REGION Network 138: CIP Line Blending Cluster 1 Request
   RUNG wire#powerrail
      Contact( "AlwaysTRUE" )
      wire#w1
      Contact( "General_Blend".Blend_Cluster1.CIP_Line1."CIP Enable" )
      Contact( "General_Blend".Blend_Cluster1.CIP_Line1."CIP Request" )
      Contact( "THE2_From_BT_To_Mixing".CIPEnable )
      wire#w2
      Coil( "Mix_to_CIP".CIP_Request."Blending Cluster 1".Blending_Cluster1_LineProduct_Request )
   END_RUNG
   RUNG wire#w1
      Contact( "General_Blend".Blend_Cluster1.CIP_Line2."CIP Enable" )
      Contact( "General_Blend".Blend_Cluster1.CIP_Line2."CIP Request" )
      Contact( "THE1_From_BT_To_Mixing".CIPEnable )
   END_RUNG wire#w2
   RUNG wire#w1
      Contact( "General_Blend".Blend_Cluster1.CIP_Line3."CIP Enable" )
      Contact( "General_Blend".Blend_Cluster1.CIP_Line3."CIP Request" )
      Contact( "General Buffer"."CIP Enable".Cluster1_Line3 )
   END_RUNG wire#w2
   // the same network as SCL:
   "Mix_to_CIP".CIP_Request."Blending Cluster 1".Blending_Cluster1_LineProduct_Request := "AlwaysTRUE" AND (("General_Blend".Blend_Cluster1.CIP_Line1."CIP Enable" AND "General_Blend".Blend_Cluster1.CIP_Line1."CIP Request" AND "THE2_From_BT_To_Mixing".CIPEnable) OR ("General_Blend".Blend_Cluster1.CIP_Line2."CIP Enable" AND "General_Blend".Blend_Cluster1.CIP_Line2."CIP Request" AND "THE1_From_BT_To_Mixing".CIPEnable) OR ("General_Blend".Blend_Cluster1.CIP_Line3."CIP Enable" AND "General_Blend".Blend_Cluster1.CIP_Line3."CIP Request" AND "General Buffer"."CIP Enable".Cluster1_Line3));
END_REGION

REGION Network 139: CIP Line Blending Cluster 1 Line OK
   RUNG wire#powerrail
      Contact( "AlwaysTRUE" )
      wire#w1
      Contact( "General_Blend".Blend_Cluster1.CIP_Line1."CIP Request" )
      Contact( "IO_Valve_Buffer_DB"."AV-22.11".FB_OPEN )
      Contact( "IO_Valve_Blend30_DB"."AV-30.12".FB_OPEN )
      wire#w2
      Contact( "IO_Valve_Blend30_DB"."AV-30.13".FB_OPEN )
      wire#w3
      Contact( "THE2_From_BT_To_Mixing".LineCIP_Open )
      wire#w4
      Coil( "Mix_to_CIP".CIP_Line_OK."Blending Cluster 1".Blending_Cluster1_LineProduct_LineOK )
   END_RUNG
   RUNG wire#w2
      Contact( "IO_Valve_Blend30_DB"."AV-30.14".FB_OPEN )
   END_RUNG wire#w3
   RUNG wire#w1
      Contact( "General_Blend".Blend_Cluster1.CIP_Line2."CIP Request" )
      Contact( "IO_Valve_Buffer_DB"."AV-22.11".FB_OPEN )
      Contact( "IO_Valve_Blend30_DB"."AV-30.15".FB_OPEN )
      wire#w5
      Contact( "IO_Valve_Blend30_DB"."AV-30.16".FB_OPEN )
      wire#w6
      Contact( "THE1_From_BT_To_Mixing".LineCIP_Open )
   END_RUNG wire#w4
   RUNG wire#w5
      Contact( "IO_Valve_Blend30_DB"."AV-30.17".FB_OPEN )
   END_RUNG wire#w6
   RUNG wire#w1
      Contact( "General_Blend".Blend_Cluster1.CIP_Line3."CIP Request" )
      Contact( "IO_Valve_Buffer_DB"."AV-22.11".FB_OPEN )
      Contact( "IO_Valve_Blend30_DB"."AV-30.18".FB_OPEN )
      wire#w7
      Contact( "IO_Valve_Blend30_DB"."AV-30.19".FB_OPEN )
      wire#w8
      Contact( "General Buffer"."CIP Line Open".Cluster1_Line3 )
   END_RUNG wire#w4
   RUNG wire#w7
      Contact( "IO_Valve_Blend30_DB"."AV-30.20".FB_OPEN )
   END_RUNG wire#w8
   // the same network as SCL:
   "Mix_to_CIP".CIP_Line_OK."Blending Cluster 1".Blending_Cluster1_LineProduct_LineOK := "AlwaysTRUE" AND (("General_Blend".Blend_Cluster1.CIP_Line1."CIP Request" AND "IO_Valve_Buffer_DB"."AV-22.11".FB_OPEN AND "IO_Valve_Blend30_DB"."AV-30.12".FB_OPEN AND ("IO_Valve_Blend30_DB"."AV-30.13".FB_OPEN OR "IO_Valve_Blend30_DB"."AV-30.14".FB_OPEN) AND "THE2_From_BT_To_Mixing".LineCIP_Open) OR ("General_Blend".Blend_Cluster1.CIP_Line2."CIP Request" AND "IO_Valve_Buffer_DB"."AV-22.11".FB_OPEN AND "IO_Valve_Blend30_DB"."AV-30.15".FB_OPEN AND ("IO_Valve_Blend30_DB"."AV-30.16".FB_OPEN OR "IO_Valve_Blend30_DB"."AV-30.17".FB_OPEN) AND "THE1_From_BT_To_Mixing".LineCIP_Open) OR ("General_Blend".Blend_Cluster1.CIP_Line3."CIP Request" AND "IO_Valve_Buffer_DB"."AV-22.11".FB_OPEN AND "IO_Valve_Blend30_DB"."AV-30.18".FB_OPEN AND ("IO_Valve_Blend30_DB"."AV-30.19".FB_OPEN OR "IO_Valve_Blend30_DB"."AV-30.20".FB_OPEN) AND "General Buffer"."CIP Line Open".Cluster1_Line3));
END_REGION

REGION Network 140: CIP Line Blending Cluster 1 Valve Cmd
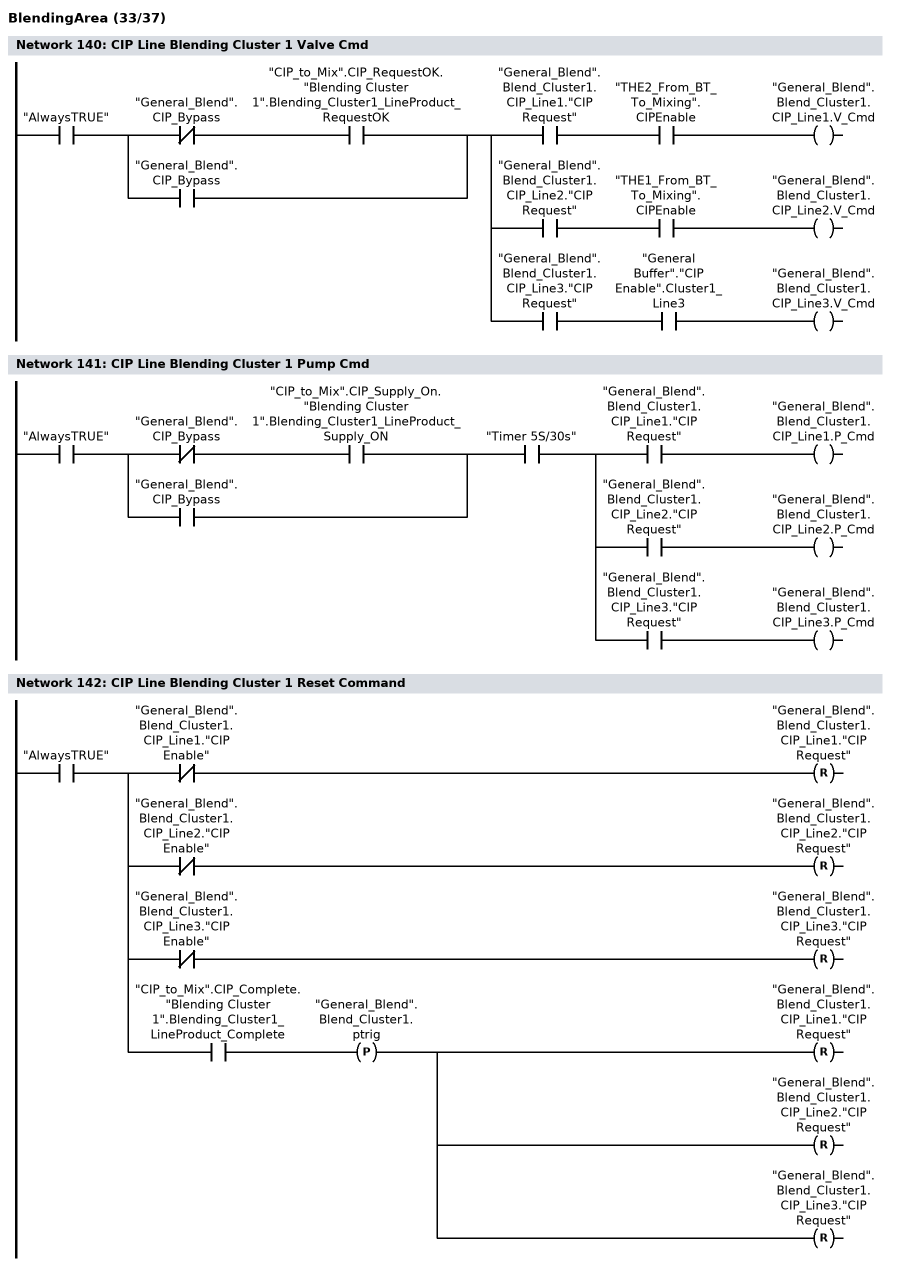
   RUNG wire#powerrail
      Contact( "AlwaysTRUE" )
      wire#w1
      I_Contact( "General_Blend".CIP_Bypass )
      Contact( "CIP_to_Mix".CIP_RequestOK."Blending Cluster 1".Blending_Cluster1_LineProduct_RequestOK )
      wire#w2
      Contact( "General_Blend".Blend_Cluster1.CIP_Line1."CIP Request" )
      Contact( "THE2_From_BT_To_Mixing".CIPEnable )
      Coil( "General_Blend".Blend_Cluster1.CIP_Line1.V_Cmd )
   END_RUNG
   RUNG wire#w1
      Contact( "General_Blend".CIP_Bypass )
   END_RUNG wire#w2
   RUNG wire#w2
      Contact( "General_Blend".Blend_Cluster1.CIP_Line2."CIP Request" )
      Contact( "THE1_From_BT_To_Mixing".CIPEnable )
      Coil( "General_Blend".Blend_Cluster1.CIP_Line2.V_Cmd )
   END_RUNG
   RUNG wire#w2
      Contact( "General_Blend".Blend_Cluster1.CIP_Line3."CIP Request" )
      Contact( "General Buffer"."CIP Enable".Cluster1_Line3 )
      Coil( "General_Blend".Blend_Cluster1.CIP_Line3.V_Cmd )
   END_RUNG
   // the same network as SCL:
   #_w1 := "AlwaysTRUE" AND ((NOT "General_Blend".CIP_Bypass AND "CIP_to_Mix".CIP_RequestOK."Blending Cluster 1".Blending_Cluster1_LineProduct_RequestOK) OR "General_Blend".CIP_Bypass);
   "General_Blend".Blend_Cluster1.CIP_Line1.V_Cmd := #_w1 AND "General_Blend".Blend_Cluster1.CIP_Line1."CIP Request" AND "THE2_From_BT_To_Mixing".CIPEnable;
   "General_Blend".Blend_Cluster1.CIP_Line2.V_Cmd := #_w1 AND "General_Blend".Blend_Cluster1.CIP_Line2."CIP Request" AND "THE1_From_BT_To_Mixing".CIPEnable;
   "General_Blend".Blend_Cluster1.CIP_Line3.V_Cmd := #_w1 AND "General_Blend".Blend_Cluster1.CIP_Line3."CIP Request" AND "General Buffer"."CIP Enable".Cluster1_Line3;
END_REGION

REGION Network 141: CIP Line Blending Cluster 1 Pump Cmd
   RUNG wire#powerrail
      Contact( "AlwaysTRUE" )
      wire#w1
      I_Contact( "General_Blend".CIP_Bypass )
      Contact( "CIP_to_Mix".CIP_Supply_On."Blending Cluster 1".Blending_Cluster1_LineProduct_Supply_ON )
      wire#w2
      Contact( "Timer 5S/30s" )
      wire#w3
      Contact( "General_Blend".Blend_Cluster1.CIP_Line1."CIP Request" )
      Coil( "General_Blend".Blend_Cluster1.CIP_Line1.P_Cmd )
   END_RUNG
   RUNG wire#w1
      Contact( "General_Blend".CIP_Bypass )
   END_RUNG wire#w2
   RUNG wire#w3
      Contact( "General_Blend".Blend_Cluster1.CIP_Line2."CIP Request" )
      Coil( "General_Blend".Blend_Cluster1.CIP_Line2.P_Cmd )
   END_RUNG
   RUNG wire#w3
      Contact( "General_Blend".Blend_Cluster1.CIP_Line3."CIP Request" )
      Coil( "General_Blend".Blend_Cluster1.CIP_Line3.P_Cmd )
   END_RUNG
   // the same network as SCL:
   #_w1 := "AlwaysTRUE" AND ((NOT "General_Blend".CIP_Bypass AND "CIP_to_Mix".CIP_Supply_On."Blending Cluster 1".Blending_Cluster1_LineProduct_Supply_ON) OR "General_Blend".CIP_Bypass) AND "Timer 5S/30s";
   "General_Blend".Blend_Cluster1.CIP_Line1.P_Cmd := #_w1 AND "General_Blend".Blend_Cluster1.CIP_Line1."CIP Request";
   "General_Blend".Blend_Cluster1.CIP_Line2.P_Cmd := #_w1 AND "General_Blend".Blend_Cluster1.CIP_Line2."CIP Request";
   "General_Blend".Blend_Cluster1.CIP_Line3.P_Cmd := #_w1 AND "General_Blend".Blend_Cluster1.CIP_Line3."CIP Request";
END_REGION

REGION Network 142: CIP Line Blending Cluster 1 Reset Command
   RUNG wire#powerrail
      Contact( "AlwaysTRUE" )
      wire#w1
      I_Contact( "General_Blend".Blend_Cluster1.CIP_Line1."CIP Enable" )
      R_Coil( "General_Blend".Blend_Cluster1.CIP_Line1."CIP Request" )
   END_RUNG
   RUNG wire#w1
      I_Contact( "General_Blend".Blend_Cluster1.CIP_Line2."CIP Enable" )
      R_Coil( "General_Blend".Blend_Cluster1.CIP_Line2."CIP Request" )
   END_RUNG
   RUNG wire#w1
      I_Contact( "General_Blend".Blend_Cluster1.CIP_Line3."CIP Enable" )
      R_Coil( "General_Blend".Blend_Cluster1.CIP_Line3."CIP Request" )
   END_RUNG
   RUNG wire#w1
      Contact( "CIP_to_Mix".CIP_Complete."Blending Cluster 1".Blending_Cluster1_LineProduct_Complete )
      P_Trig( "General_Blend".Blend_Cluster1.ptrig )
      wire#w2
      R_Coil( "General_Blend".Blend_Cluster1.CIP_Line1."CIP Request" )
   END_RUNG
   RUNG wire#w2
      R_Coil( "General_Blend".Blend_Cluster1.CIP_Line2."CIP Request" )
   END_RUNG
   RUNG wire#w2
      R_Coil( "General_Blend".Blend_Cluster1.CIP_Line3."CIP Request" )
   END_RUNG
   // the same network as SCL:
   IF "AlwaysTRUE" AND NOT "General_Blend".Blend_Cluster1.CIP_Line1."CIP Enable" THEN
       "General_Blend".Blend_Cluster1.CIP_Line1."CIP Request" := FALSE;
   END_IF;
   IF "AlwaysTRUE" AND NOT "General_Blend".Blend_Cluster1.CIP_Line2."CIP Enable" THEN
       "General_Blend".Blend_Cluster1.CIP_Line2."CIP Request" := FALSE;
   END_IF;
   IF "AlwaysTRUE" AND NOT "General_Blend".Blend_Cluster1.CIP_Line3."CIP Enable" THEN
       "General_Blend".Blend_Cluster1.CIP_Line3."CIP Request" := FALSE;
   END_IF;
   #_w1 := "AlwaysTRUE" AND "CIP_to_Mix".CIP_Complete."Blending Cluster 1".Blending_Cluster1_LineProduct_Complete;
   #_w2 := #_w1 AND NOT "General_Blend".Blend_Cluster1.ptrig;   // rising edge
   "General_Blend".Blend_Cluster1.ptrig := #_w1;
   IF #_w2 THEN
       "General_Blend".Blend_Cluster1.CIP_Line1."CIP Request" := FALSE;
       "General_Blend".Blend_Cluster1.CIP_Line2."CIP Request" := FALSE;
       "General_Blend".Blend_Cluster1.CIP_Line3."CIP Request" := FALSE;
   END_IF;
END_REGION

REGION Network 144: CIP Line Blending Cluster 2 Enable
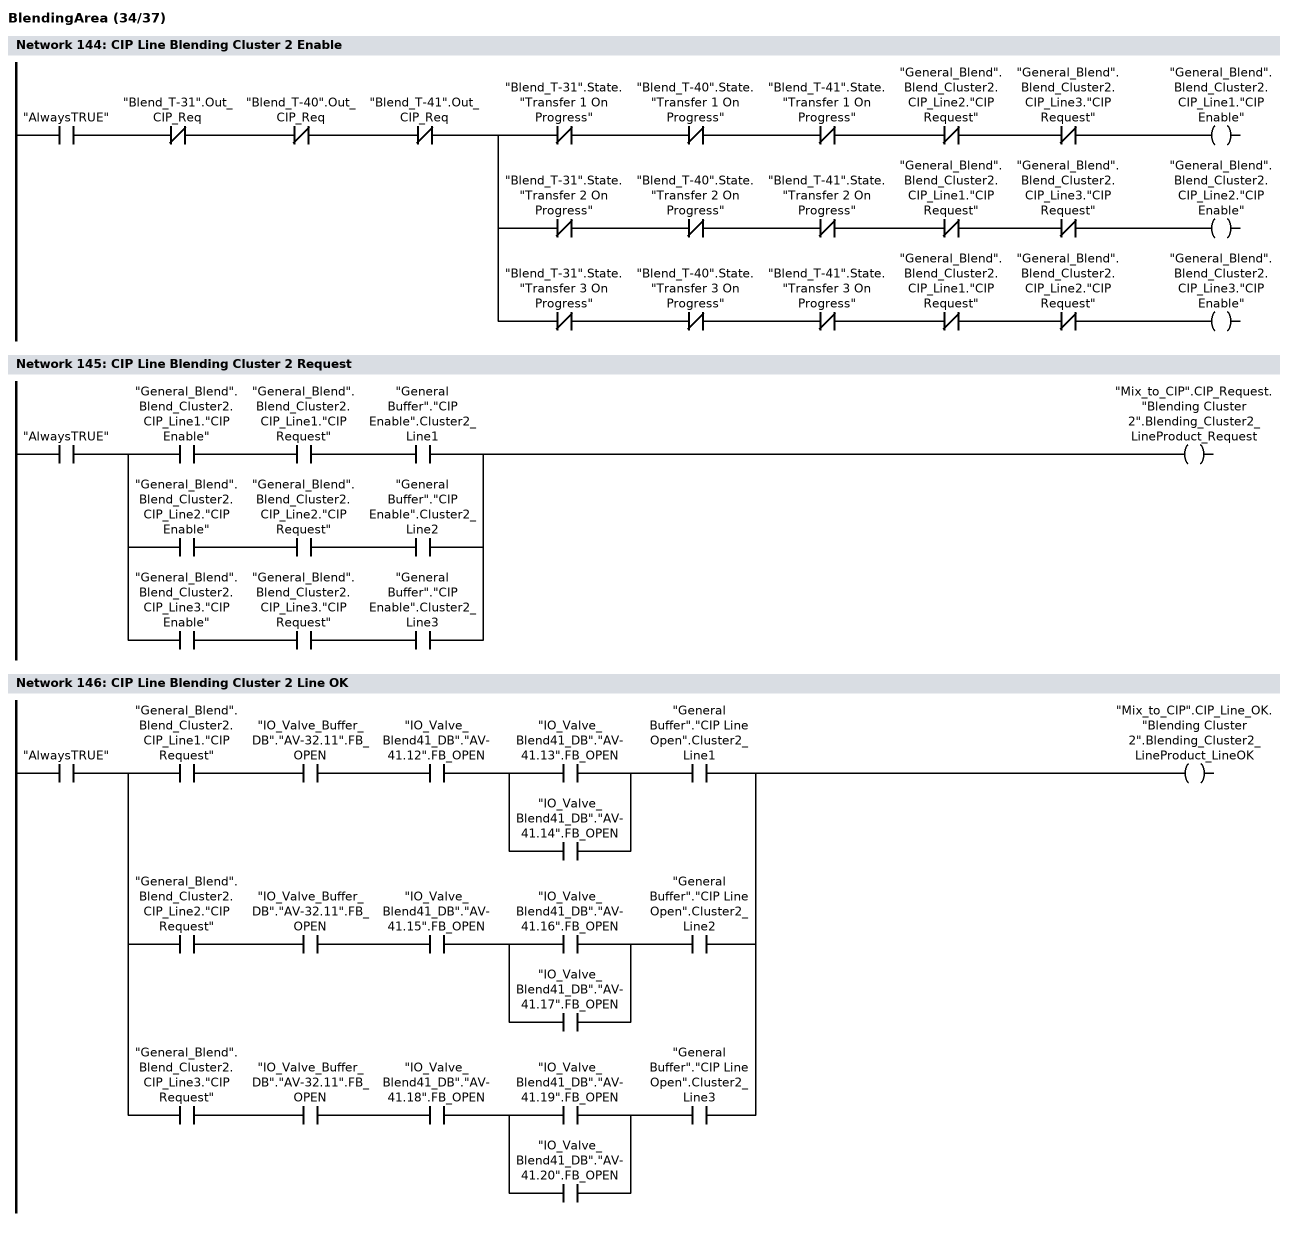
   RUNG wire#powerrail
      Contact( "AlwaysTRUE" )
      I_Contact( "Blend_T-31".Out_CIP_Req )
      I_Contact( "Blend_T-40".Out_CIP_Req )
      I_Contact( "Blend_T-41".Out_CIP_Req )
      wire#w1
      I_Contact( "Blend_T-31".State."Transfer 1 On Progress" )
      I_Contact( "Blend_T-40".State."Transfer 1 On Progress" )
      I_Contact( "Blend_T-41".State."Transfer 1 On Progress" )
      I_Contact( "General_Blend".Blend_Cluster2.CIP_Line2."CIP Request" )
      I_Contact( "General_Blend".Blend_Cluster2.CIP_Line3."CIP Request" )
      Coil( "General_Blend".Blend_Cluster2.CIP_Line1."CIP Enable" )
   END_RUNG
   RUNG wire#w1
      I_Contact( "Blend_T-31".State."Transfer 2 On Progress" )
      I_Contact( "Blend_T-40".State."Transfer 2 On Progress" )
      I_Contact( "Blend_T-41".State."Transfer 2 On Progress" )
      I_Contact( "General_Blend".Blend_Cluster2.CIP_Line1."CIP Request" )
      I_Contact( "General_Blend".Blend_Cluster2.CIP_Line3."CIP Request" )
      Coil( "General_Blend".Blend_Cluster2.CIP_Line2."CIP Enable" )
   END_RUNG
   RUNG wire#w1
      I_Contact( "Blend_T-31".State."Transfer 3 On Progress" )
      I_Contact( "Blend_T-40".State."Transfer 3 On Progress" )
      I_Contact( "Blend_T-41".State."Transfer 3 On Progress" )
      I_Contact( "General_Blend".Blend_Cluster2.CIP_Line1."CIP Request" )
      I_Contact( "General_Blend".Blend_Cluster2.CIP_Line2."CIP Request" )
      Coil( "General_Blend".Blend_Cluster2.CIP_Line3."CIP Enable" )
   END_RUNG
   // the same network as SCL:
   #_w1 := "AlwaysTRUE" AND NOT "Blend_T-31".Out_CIP_Req AND NOT "Blend_T-40".Out_CIP_Req AND NOT "Blend_T-41".Out_CIP_Req;
   "General_Blend".Blend_Cluster2.CIP_Line1."CIP Enable" := #_w1 AND NOT "Blend_T-31".State."Transfer 1 On Progress" AND NOT "Blend_T-40".State."Transfer 1 On Progress" AND NOT "Blend_T-41".State."Transfer 1 On Progress" AND NOT "General_Blend".Blend_Cluster2.CIP_Line2."CIP Request" AND NOT "General_Blend".Blend_Cluster2.CIP_Line3."CIP Request";
   "General_Blend".Blend_Cluster2.CIP_Line2."CIP Enable" := #_w1 AND NOT "Blend_T-31".State."Transfer 2 On Progress" AND NOT "Blend_T-40".State."Transfer 2 On Progress" AND NOT "Blend_T-41".State."Transfer 2 On Progress" AND NOT "General_Blend".Blend_Cluster2.CIP_Line1."CIP Request" AND NOT "General_Blend".Blend_Cluster2.CIP_Line3."CIP Request";
   "General_Blend".Blend_Cluster2.CIP_Line3."CIP Enable" := #_w1 AND NOT "Blend_T-31".State."Transfer 3 On Progress" AND NOT "Blend_T-40".State."Transfer 3 On Progress" AND NOT "Blend_T-41".State."Transfer 3 On Progress" AND NOT "General_Blend".Blend_Cluster2.CIP_Line1."CIP Request" AND NOT "General_Blend".Blend_Cluster2.CIP_Line2."CIP Request";
END_REGION

REGION Network 145: CIP Line Blending Cluster 2 Request
   RUNG wire#powerrail
      Contact( "AlwaysTRUE" )
      wire#w1
      Contact( "General_Blend".Blend_Cluster2.CIP_Line1."CIP Enable" )
      Contact( "General_Blend".Blend_Cluster2.CIP_Line1."CIP Request" )
      Contact( "General Buffer"."CIP Enable".Cluster2_Line1 )
      wire#w2
      Coil( "Mix_to_CIP".CIP_Request."Blending Cluster 2".Blending_Cluster2_LineProduct_Request )
   END_RUNG
   RUNG wire#w1
      Contact( "General_Blend".Blend_Cluster2.CIP_Line2."CIP Enable" )
      Contact( "General_Blend".Blend_Cluster2.CIP_Line2."CIP Request" )
      Contact( "General Buffer"."CIP Enable".Cluster2_Line2 )
   END_RUNG wire#w2
   RUNG wire#w1
      Contact( "General_Blend".Blend_Cluster2.CIP_Line3."CIP Enable" )
      Contact( "General_Blend".Blend_Cluster2.CIP_Line3."CIP Request" )
      Contact( "General Buffer"."CIP Enable".Cluster2_Line3 )
   END_RUNG wire#w2
   // the same network as SCL:
   "Mix_to_CIP".CIP_Request."Blending Cluster 2".Blending_Cluster2_LineProduct_Request := "AlwaysTRUE" AND (("General_Blend".Blend_Cluster2.CIP_Line1."CIP Enable" AND "General_Blend".Blend_Cluster2.CIP_Line1."CIP Request" AND "General Buffer"."CIP Enable".Cluster2_Line1) OR ("General_Blend".Blend_Cluster2.CIP_Line2."CIP Enable" AND "General_Blend".Blend_Cluster2.CIP_Line2."CIP Request" AND "General Buffer"."CIP Enable".Cluster2_Line2) OR ("General_Blend".Blend_Cluster2.CIP_Line3."CIP Enable" AND "General_Blend".Blend_Cluster2.CIP_Line3."CIP Request" AND "General Buffer"."CIP Enable".Cluster2_Line3));
END_REGION

REGION Network 146: CIP Line Blending Cluster 2 Line OK
   RUNG wire#powerrail
      Contact( "AlwaysTRUE" )
      wire#w1
      Contact( "General_Blend".Blend_Cluster2.CIP_Line1."CIP Request" )
      Contact( "IO_Valve_Buffer_DB"."AV-32.11".FB_OPEN )
      Contact( "IO_Valve_Blend41_DB"."AV-41.12".FB_OPEN )
      wire#w2
      Contact( "IO_Valve_Blend41_DB"."AV-41.13".FB_OPEN )
      wire#w3
      Contact( "General Buffer"."CIP Line Open".Cluster2_Line1 )
      wire#w4
      Coil( "Mix_to_CIP".CIP_Line_OK."Blending Cluster 2".Blending_Cluster2_LineProduct_LineOK )
   END_RUNG
   RUNG wire#w2
      Contact( "IO_Valve_Blend41_DB"."AV-41.14".FB_OPEN )
   END_RUNG wire#w3
   RUNG wire#w1
      Contact( "General_Blend".Blend_Cluster2.CIP_Line2."CIP Request" )
      Contact( "IO_Valve_Buffer_DB"."AV-32.11".FB_OPEN )
      Contact( "IO_Valve_Blend41_DB"."AV-41.15".FB_OPEN )
      wire#w5
      Contact( "IO_Valve_Blend41_DB"."AV-41.16".FB_OPEN )
      wire#w6
      Contact( "General Buffer"."CIP Line Open".Cluster2_Line2 )
   END_RUNG wire#w4
   RUNG wire#w5
      Contact( "IO_Valve_Blend41_DB"."AV-41.17".FB_OPEN )
   END_RUNG wire#w6
   RUNG wire#w1
      Contact( "General_Blend".Blend_Cluster2.CIP_Line3."CIP Request" )
      Contact( "IO_Valve_Buffer_DB"."AV-32.11".FB_OPEN )
      Contact( "IO_Valve_Blend41_DB"."AV-41.18".FB_OPEN )
      wire#w7
      Contact( "IO_Valve_Blend41_DB"."AV-41.19".FB_OPEN )
      wire#w8
      Contact( "General Buffer"."CIP Line Open".Cluster2_Line3 )
   END_RUNG wire#w4
   RUNG wire#w7
      Contact( "IO_Valve_Blend41_DB"."AV-41.20".FB_OPEN )
   END_RUNG wire#w8
   // the same network as SCL:
   "Mix_to_CIP".CIP_Line_OK."Blending Cluster 2".Blending_Cluster2_LineProduct_LineOK := "AlwaysTRUE" AND (("General_Blend".Blend_Cluster2.CIP_Line1."CIP Request" AND "IO_Valve_Buffer_DB"."AV-32.11".FB_OPEN AND "IO_Valve_Blend41_DB"."AV-41.12".FB_OPEN AND ("IO_Valve_Blend41_DB"."AV-41.13".FB_OPEN OR "IO_Valve_Blend41_DB"."AV-41.14".FB_OPEN) AND "General Buffer"."CIP Line Open".Cluster2_Line1) OR ("General_Blend".Blend_Cluster2.CIP_Line2."CIP Request" AND "IO_Valve_Buffer_DB"."AV-32.11".FB_OPEN AND "IO_Valve_Blend41_DB"."AV-41.15".FB_OPEN AND ("IO_Valve_Blend41_DB"."AV-41.16".FB_OPEN OR "IO_Valve_Blend41_DB"."AV-41.17".FB_OPEN) AND "General Buffer"."CIP Line Open".Cluster2_Line2) OR ("General_Blend".Blend_Cluster2.CIP_Line3."CIP Request" AND "IO_Valve_Buffer_DB"."AV-32.11".FB_OPEN AND "IO_Valve_Blend41_DB"."AV-41.18".FB_OPEN AND ("IO_Valve_Blend41_DB"."AV-41.19".FB_OPEN OR "IO_Valve_Blend41_DB"."AV-41.20".FB_OPEN) AND "General Buffer"."CIP Line Open".Cluster2_Line3));
END_REGION

REGION Network 147: CIP Line Blending Cluster 2 Valve Cmd
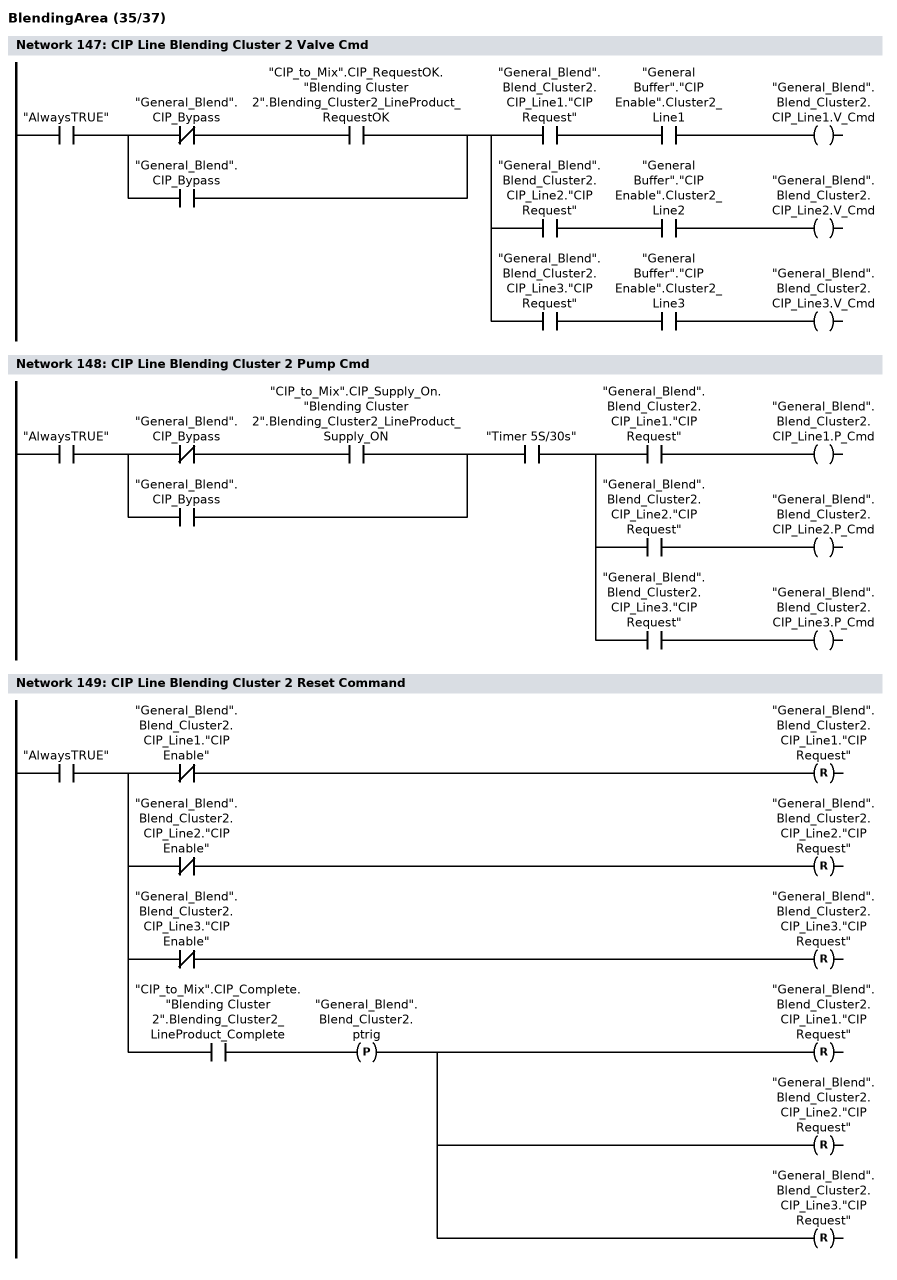
   RUNG wire#powerrail
      Contact( "AlwaysTRUE" )
      wire#w1
      I_Contact( "General_Blend".CIP_Bypass )
      Contact( "CIP_to_Mix".CIP_RequestOK."Blending Cluster 2".Blending_Cluster2_LineProduct_RequestOK )
      wire#w2
      Contact( "General_Blend".Blend_Cluster2.CIP_Line1."CIP Request" )
      Contact( "General Buffer"."CIP Enable".Cluster2_Line1 )
      Coil( "General_Blend".Blend_Cluster2.CIP_Line1.V_Cmd )
   END_RUNG
   RUNG wire#w1
      Contact( "General_Blend".CIP_Bypass )
   END_RUNG wire#w2
   RUNG wire#w2
      Contact( "General_Blend".Blend_Cluster2.CIP_Line2."CIP Request" )
      Contact( "General Buffer"."CIP Enable".Cluster2_Line2 )
      Coil( "General_Blend".Blend_Cluster2.CIP_Line2.V_Cmd )
   END_RUNG
   RUNG wire#w2
      Contact( "General_Blend".Blend_Cluster2.CIP_Line3."CIP Request" )
      Contact( "General Buffer"."CIP Enable".Cluster2_Line3 )
      Coil( "General_Blend".Blend_Cluster2.CIP_Line3.V_Cmd )
   END_RUNG
   // the same network as SCL:
   #_w1 := "AlwaysTRUE" AND ((NOT "General_Blend".CIP_Bypass AND "CIP_to_Mix".CIP_RequestOK."Blending Cluster 2".Blending_Cluster2_LineProduct_RequestOK) OR "General_Blend".CIP_Bypass);
   "General_Blend".Blend_Cluster2.CIP_Line1.V_Cmd := #_w1 AND "General_Blend".Blend_Cluster2.CIP_Line1."CIP Request" AND "General Buffer"."CIP Enable".Cluster2_Line1;
   "General_Blend".Blend_Cluster2.CIP_Line2.V_Cmd := #_w1 AND "General_Blend".Blend_Cluster2.CIP_Line2."CIP Request" AND "General Buffer"."CIP Enable".Cluster2_Line2;
   "General_Blend".Blend_Cluster2.CIP_Line3.V_Cmd := #_w1 AND "General_Blend".Blend_Cluster2.CIP_Line3."CIP Request" AND "General Buffer"."CIP Enable".Cluster2_Line3;
END_REGION

REGION Network 148: CIP Line Blending Cluster 2 Pump Cmd
   RUNG wire#powerrail
      Contact( "AlwaysTRUE" )
      wire#w1
      I_Contact( "General_Blend".CIP_Bypass )
      Contact( "CIP_to_Mix".CIP_Supply_On."Blending Cluster 2".Blending_Cluster2_LineProduct_Supply_ON )
      wire#w2
      Contact( "Timer 5S/30s" )
      wire#w3
      Contact( "General_Blend".Blend_Cluster2.CIP_Line1."CIP Request" )
      Coil( "General_Blend".Blend_Cluster2.CIP_Line1.P_Cmd )
   END_RUNG
   RUNG wire#w1
      Contact( "General_Blend".CIP_Bypass )
   END_RUNG wire#w2
   RUNG wire#w3
      Contact( "General_Blend".Blend_Cluster2.CIP_Line2."CIP Request" )
      Coil( "General_Blend".Blend_Cluster2.CIP_Line2.P_Cmd )
   END_RUNG
   RUNG wire#w3
      Contact( "General_Blend".Blend_Cluster2.CIP_Line3."CIP Request" )
      Coil( "General_Blend".Blend_Cluster2.CIP_Line3.P_Cmd )
   END_RUNG
   // the same network as SCL:
   #_w1 := "AlwaysTRUE" AND ((NOT "General_Blend".CIP_Bypass AND "CIP_to_Mix".CIP_Supply_On."Blending Cluster 2".Blending_Cluster2_LineProduct_Supply_ON) OR "General_Blend".CIP_Bypass) AND "Timer 5S/30s";
   "General_Blend".Blend_Cluster2.CIP_Line1.P_Cmd := #_w1 AND "General_Blend".Blend_Cluster2.CIP_Line1."CIP Request";
   "General_Blend".Blend_Cluster2.CIP_Line2.P_Cmd := #_w1 AND "General_Blend".Blend_Cluster2.CIP_Line2."CIP Request";
   "General_Blend".Blend_Cluster2.CIP_Line3.P_Cmd := #_w1 AND "General_Blend".Blend_Cluster2.CIP_Line3."CIP Request";
END_REGION

REGION Network 149: CIP Line Blending Cluster 2 Reset Command
   RUNG wire#powerrail
      Contact( "AlwaysTRUE" )
      wire#w1
      I_Contact( "General_Blend".Blend_Cluster2.CIP_Line1."CIP Enable" )
      R_Coil( "General_Blend".Blend_Cluster2.CIP_Line1."CIP Request" )
   END_RUNG
   RUNG wire#w1
      I_Contact( "General_Blend".Blend_Cluster2.CIP_Line2."CIP Enable" )
      R_Coil( "General_Blend".Blend_Cluster2.CIP_Line2."CIP Request" )
   END_RUNG
   RUNG wire#w1
      I_Contact( "General_Blend".Blend_Cluster2.CIP_Line3."CIP Enable" )
      R_Coil( "General_Blend".Blend_Cluster2.CIP_Line3."CIP Request" )
   END_RUNG
   RUNG wire#w1
      Contact( "CIP_to_Mix".CIP_Complete."Blending Cluster 2".Blending_Cluster2_LineProduct_Complete )
      P_Trig( "General_Blend".Blend_Cluster2.ptrig )
      wire#w2
      R_Coil( "General_Blend".Blend_Cluster2.CIP_Line1."CIP Request" )
   END_RUNG
   RUNG wire#w2
      R_Coil( "General_Blend".Blend_Cluster2.CIP_Line2."CIP Request" )
   END_RUNG
   RUNG wire#w2
      R_Coil( "General_Blend".Blend_Cluster2.CIP_Line3."CIP Request" )
   END_RUNG
   // the same network as SCL:
   IF "AlwaysTRUE" AND NOT "General_Blend".Blend_Cluster2.CIP_Line1."CIP Enable" THEN
       "General_Blend".Blend_Cluster2.CIP_Line1."CIP Request" := FALSE;
   END_IF;
   IF "AlwaysTRUE" AND NOT "General_Blend".Blend_Cluster2.CIP_Line2."CIP Enable" THEN
       "General_Blend".Blend_Cluster2.CIP_Line2."CIP Request" := FALSE;
   END_IF;
   IF "AlwaysTRUE" AND NOT "General_Blend".Blend_Cluster2.CIP_Line3."CIP Enable" THEN
       "General_Blend".Blend_Cluster2.CIP_Line3."CIP Request" := FALSE;
   END_IF;
   #_w1 := "AlwaysTRUE" AND "CIP_to_Mix".CIP_Complete."Blending Cluster 2".Blending_Cluster2_LineProduct_Complete;
   #_w2 := #_w1 AND NOT "General_Blend".Blend_Cluster2.ptrig;   // rising edge
   "General_Blend".Blend_Cluster2.ptrig := #_w1;
   IF #_w2 THEN
       "General_Blend".Blend_Cluster2.CIP_Line1."CIP Request" := FALSE;
       "General_Blend".Blend_Cluster2.CIP_Line2."CIP Request" := FALSE;
       "General_Blend".Blend_Cluster2.CIP_Line3."CIP Request" := FALSE;
   END_IF;
END_REGION

REGION Network 151: CIP to Return Line 1
   // Only for Blend Tank, Because CIP Supply from line 2 while Blend Tank can choose to return through line 1 or 2
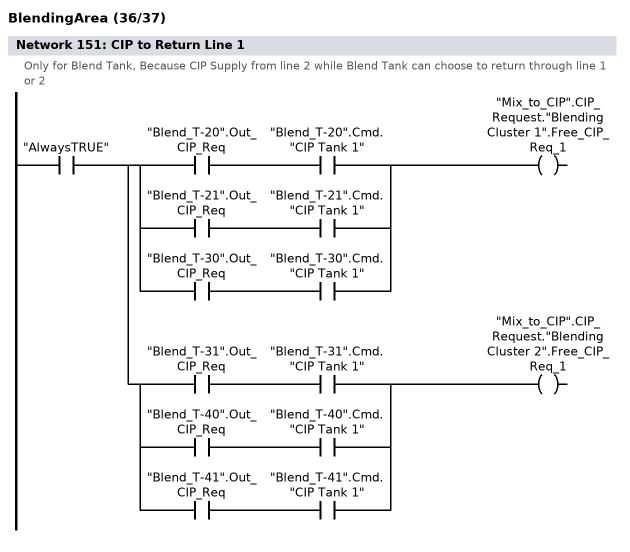
   RUNG wire#powerrail
      Contact( "AlwaysTRUE" )
      wire#w1
      Contact( "Blend_T-20".Out_CIP_Req )
      Contact( "Blend_T-20".Cmd."CIP Tank 1" )
      wire#w2
      Coil( "Mix_to_CIP".CIP_Request."Blending Cluster 1".Free_CIP_Req_1 )
   END_RUNG
   RUNG wire#w1
      Contact( "Blend_T-21".Out_CIP_Req )
      Contact( "Blend_T-21".Cmd."CIP Tank 1" )
   END_RUNG wire#w2
   RUNG wire#w1
      Contact( "Blend_T-30".Out_CIP_Req )
      Contact( "Blend_T-30".Cmd."CIP Tank 1" )
   END_RUNG wire#w2
   RUNG wire#w1
      Contact( "Blend_T-31".Out_CIP_Req )
      Contact( "Blend_T-31".Cmd."CIP Tank 1" )
      wire#w3
      Coil( "Mix_to_CIP".CIP_Request."Blending Cluster 2".Free_CIP_Req_1 )
   END_RUNG
   RUNG wire#w1
      Contact( "Blend_T-40".Out_CIP_Req )
      Contact( "Blend_T-40".Cmd."CIP Tank 1" )
   END_RUNG wire#w3
   RUNG wire#w1
      Contact( "Blend_T-41".Out_CIP_Req )
      Contact( "Blend_T-41".Cmd."CIP Tank 1" )
   END_RUNG wire#w3
   // the same network as SCL:
   "Mix_to_CIP".CIP_Request."Blending Cluster 1".Free_CIP_Req_1 := "AlwaysTRUE" AND (("Blend_T-20".Out_CIP_Req AND "Blend_T-20".Cmd."CIP Tank 1") OR ("Blend_T-21".Out_CIP_Req AND "Blend_T-21".Cmd."CIP Tank 1") OR ("Blend_T-30".Out_CIP_Req AND "Blend_T-30".Cmd."CIP Tank 1"));
   "Mix_to_CIP".CIP_Request."Blending Cluster 2".Free_CIP_Req_1 := "AlwaysTRUE" AND (("Blend_T-31".Out_CIP_Req AND "Blend_T-31".Cmd."CIP Tank 1") OR ("Blend_T-40".Out_CIP_Req AND "Blend_T-40".Cmd."CIP Tank 1") OR ("Blend_T-41".Out_CIP_Req AND "Blend_T-41".Cmd."CIP Tank 1"));
END_REGION

REGION Network 153: Valve
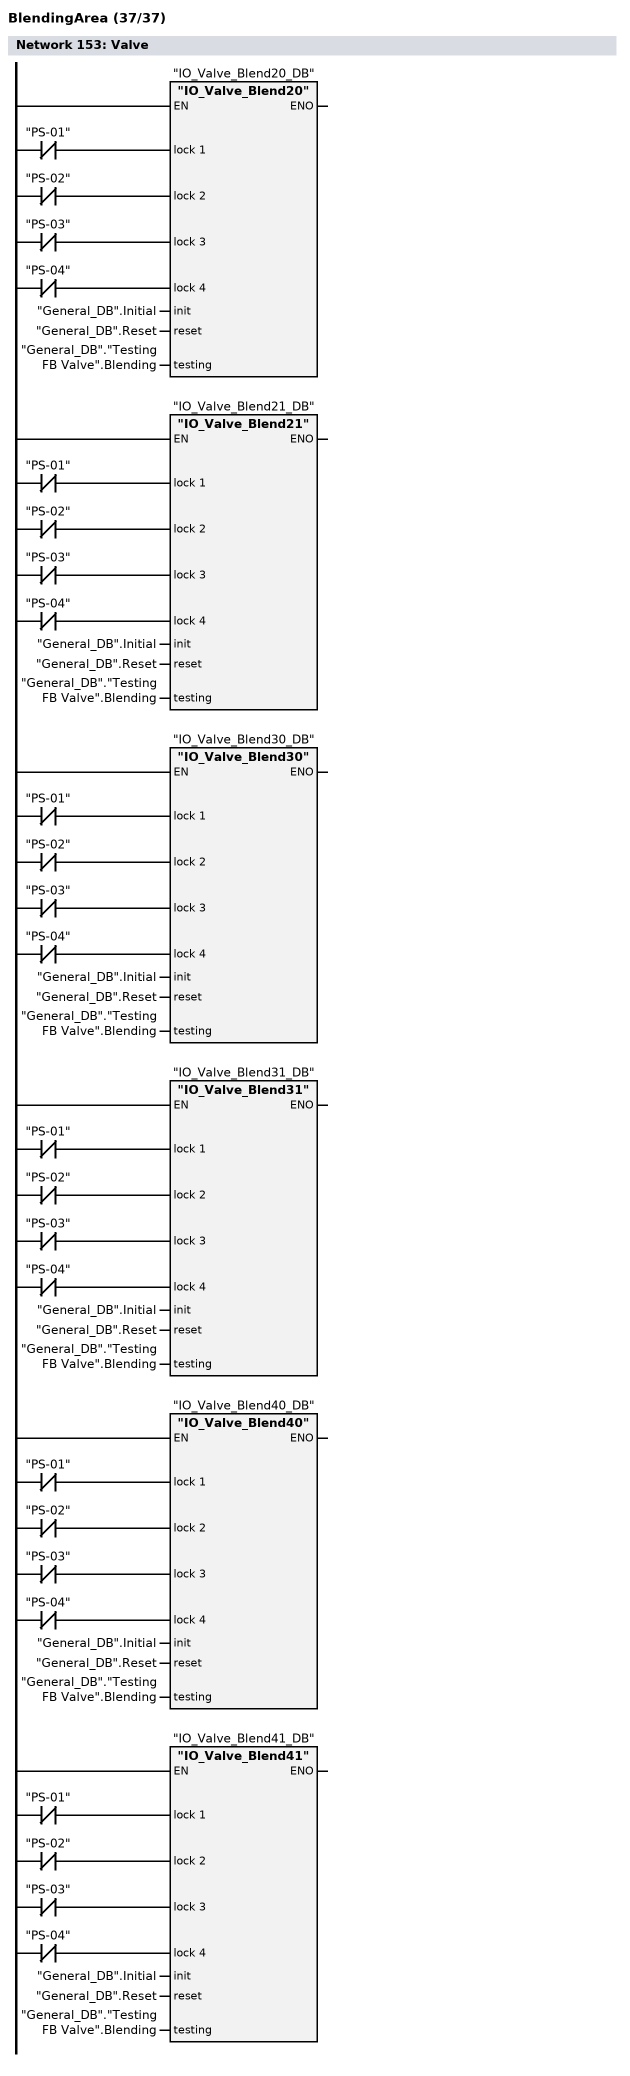
   RUNG wire#powerrail
      "IO_Valve_Blend20_DB"("lock 1" := wire#w1, "lock 2" := wire#w2, "lock 3" := wire#w3, "lock 4" := wire#w4, init := "General_DB".Initial, reset := "General_DB".Reset, testing := "General_DB"."Testing FB Valve".Blending)
   END_RUNG
   RUNG wire#powerrail
      I_Contact( "PS-01" )
   END_RUNG wire#w1
   RUNG wire#powerrail
      I_Contact( "PS-02" )
   END_RUNG wire#w2
   RUNG wire#powerrail
      I_Contact( "PS-03" )
   END_RUNG wire#w3
   RUNG wire#powerrail
      I_Contact( "PS-04" )
   END_RUNG wire#w4
   RUNG wire#powerrail
      "IO_Valve_Blend21_DB"("lock 1" := wire#w5, "lock 2" := wire#w6, "lock 3" := wire#w7, "lock 4" := wire#w8, init := "General_DB".Initial, reset := "General_DB".Reset, testing := "General_DB"."Testing FB Valve".Blending)
   END_RUNG
   RUNG wire#powerrail
      I_Contact( "PS-01" )
   END_RUNG wire#w5
   RUNG wire#powerrail
      I_Contact( "PS-02" )
   END_RUNG wire#w6
   RUNG wire#powerrail
      I_Contact( "PS-03" )
   END_RUNG wire#w7
   RUNG wire#powerrail
      I_Contact( "PS-04" )
   END_RUNG wire#w8
   RUNG wire#powerrail
      "IO_Valve_Blend30_DB"("lock 1" := wire#w9, "lock 2" := wire#w10, "lock 3" := wire#w11, "lock 4" := wire#w12, init := "General_DB".Initial, reset := "General_DB".Reset, testing := "General_DB"."Testing FB Valve".Blending)
   END_RUNG
   RUNG wire#powerrail
      I_Contact( "PS-01" )
   END_RUNG wire#w9
   RUNG wire#powerrail
      I_Contact( "PS-02" )
   END_RUNG wire#w10
   RUNG wire#powerrail
      I_Contact( "PS-03" )
   END_RUNG wire#w11
   RUNG wire#powerrail
      I_Contact( "PS-04" )
   END_RUNG wire#w12
   RUNG wire#powerrail
      "IO_Valve_Blend31_DB"("lock 1" := wire#w13, "lock 2" := wire#w14, "lock 3" := wire#w15, "lock 4" := wire#w16, init := "General_DB".Initial, reset := "General_DB".Reset, testing := "General_DB"."Testing FB Valve".Blending)
   END_RUNG
   RUNG wire#powerrail
      I_Contact( "PS-01" )
   END_RUNG wire#w13
   RUNG wire#powerrail
      I_Contact( "PS-02" )
   END_RUNG wire#w14
   RUNG wire#powerrail
      I_Contact( "PS-03" )
   END_RUNG wire#w15
   RUNG wire#powerrail
      I_Contact( "PS-04" )
   END_RUNG wire#w16
   RUNG wire#powerrail
      "IO_Valve_Blend40_DB"("lock 1" := wire#w17, "lock 2" := wire#w18, "lock 3" := wire#w19, "lock 4" := wire#w20, init := "General_DB".Initial, reset := "General_DB".Reset, testing := "General_DB"."Testing FB Valve".Blending)
   END_RUNG
   RUNG wire#powerrail
      I_Contact( "PS-01" )
   END_RUNG wire#w17
   RUNG wire#powerrail
      I_Contact( "PS-02" )
   END_RUNG wire#w18
   RUNG wire#powerrail
      I_Contact( "PS-03" )
   END_RUNG wire#w19
   RUNG wire#powerrail
      I_Contact( "PS-04" )
   END_RUNG wire#w20
   RUNG wire#powerrail
      "IO_Valve_Blend41_DB"("lock 1" := wire#w21, "lock 2" := wire#w22, "lock 3" := wire#w23, "lock 4" := wire#w24, init := "General_DB".Initial, reset := "General_DB".Reset, testing := "General_DB"."Testing FB Valve".Blending)
   END_RUNG
   RUNG wire#powerrail
      I_Contact( "PS-01" )
   END_RUNG wire#w21
   RUNG wire#powerrail
      I_Contact( "PS-02" )
   END_RUNG wire#w22
   RUNG wire#powerrail
      I_Contact( "PS-03" )
   END_RUNG wire#w23
   RUNG wire#powerrail
      I_Contact( "PS-04" )
   END_RUNG wire#w24
   // the same network as SCL:
   "IO_Valve_Blend20_DB"("lock 1" := NOT "PS-01",   // "IO_Valve_Blend20"
                         "lock 2" := NOT "PS-02",
                         "lock 3" := NOT "PS-03",
                         "lock 4" := NOT "PS-04",
                         init := "General_DB".Initial,
                         reset := "General_DB".Reset,
                         testing := "General_DB"."Testing FB Valve".Blending);
   "IO_Valve_Blend21_DB"("lock 1" := NOT "PS-01",   // "IO_Valve_Blend21"
                         "lock 2" := NOT "PS-02",
                         "lock 3" := NOT "PS-03",
                         "lock 4" := NOT "PS-04",
                         init := "General_DB".Initial,
                         reset := "General_DB".Reset,
                         testing := "General_DB"."Testing FB Valve".Blending);
   "IO_Valve_Blend30_DB"("lock 1" := NOT "PS-01",   // "IO_Valve_Blend30"
                         "lock 2" := NOT "PS-02",
                         "lock 3" := NOT "PS-03",
                         "lock 4" := NOT "PS-04",
                         init := "General_DB".Initial,
                         reset := "General_DB".Reset,
                         testing := "General_DB"."Testing FB Valve".Blending);
   "IO_Valve_Blend31_DB"("lock 1" := NOT "PS-01",   // "IO_Valve_Blend31"
                         "lock 2" := NOT "PS-02",
                         "lock 3" := NOT "PS-03",
                         "lock 4" := NOT "PS-04",
                         init := "General_DB".Initial,
                         reset := "General_DB".Reset,
                         testing := "General_DB"."Testing FB Valve".Blending);
   "IO_Valve_Blend40_DB"("lock 1" := NOT "PS-01",   // "IO_Valve_Blend40"
                         "lock 2" := NOT "PS-02",
                         "lock 3" := NOT "PS-03",
                         "lock 4" := NOT "PS-04",
                         init := "General_DB".Initial,
                         reset := "General_DB".Reset,
                         testing := "General_DB"."Testing FB Valve".Blending);
   "IO_Valve_Blend41_DB"("lock 1" := NOT "PS-01",   // "IO_Valve_Blend41"
                         "lock 2" := NOT "PS-02",
                         "lock 3" := NOT "PS-03",
                         "lock 4" := NOT "PS-04",
                         init := "General_DB".Initial,
                         reset := "General_DB".Reset,
                         testing := "General_DB"."Testing FB Valve".Blending);
END_REGION
END_FUNCTION

FUNCTION_BLOCK "IO Analog Blending"   // FB10, LAD
{ S7_Optimized_Access := 'FALSE' }
VERSION : 0.1
// stored: AutoNumber true, IsIECCheckEnabled false, SetENOAutomatically false, UDAEnableTagReadback false
   VAR_INPUT
      Init : Bool;
      Reset : Bool;
   END_VAR
   VAR
      "LT-20.01" { S7_SetPoint := 'True'} : "Ana_w_K1K2";
      "LT-21.01" { S7_SetPoint := 'True'} : "Ana_w_K1K2";
      "LT-22.01" { S7_SetPoint := 'True'} : "Ana_w_K1K2";
      "LT-30.01" { S7_SetPoint := 'True'} : "Ana_w_K1K2";
      "LT-31.01" { S7_SetPoint := 'True'} : "Ana_w_K1K2";
      "LT-32.01" { S7_SetPoint := 'True'} : "Ana_w_K1K2";
      "FT-15.01" { S7_SetPoint := 'True'} : "Ana_w_K1K2";
      "FT-15.01Com" { S7_SetPoint := 'True'} : "Read FT Comm";
      "FT-22.01" { S7_SetPoint := 'True'} : "Ana_w_K1K2";
      "FT-22.01Com" { S7_SetPoint := 'True'} : "Read FT Comm";
      "FT-32.01" { S7_SetPoint := 'True'} : "Ana_w_K1K2";
      "FT-32.01Com" { S7_SetPoint := 'True'} : "Read FT Comm";
      "LT-40.01" { S7_SetPoint := 'True'} : "Ana_w_K1K2";
      "LT-41.01" { S7_SetPoint := 'True'} : "Ana_w_K1K2";
      "FT-00.01" { S7_SetPoint := 'True'} : "Ana_w_K1K2";
   END_VAR
BEGIN

REGION Network 1: LT-20.01
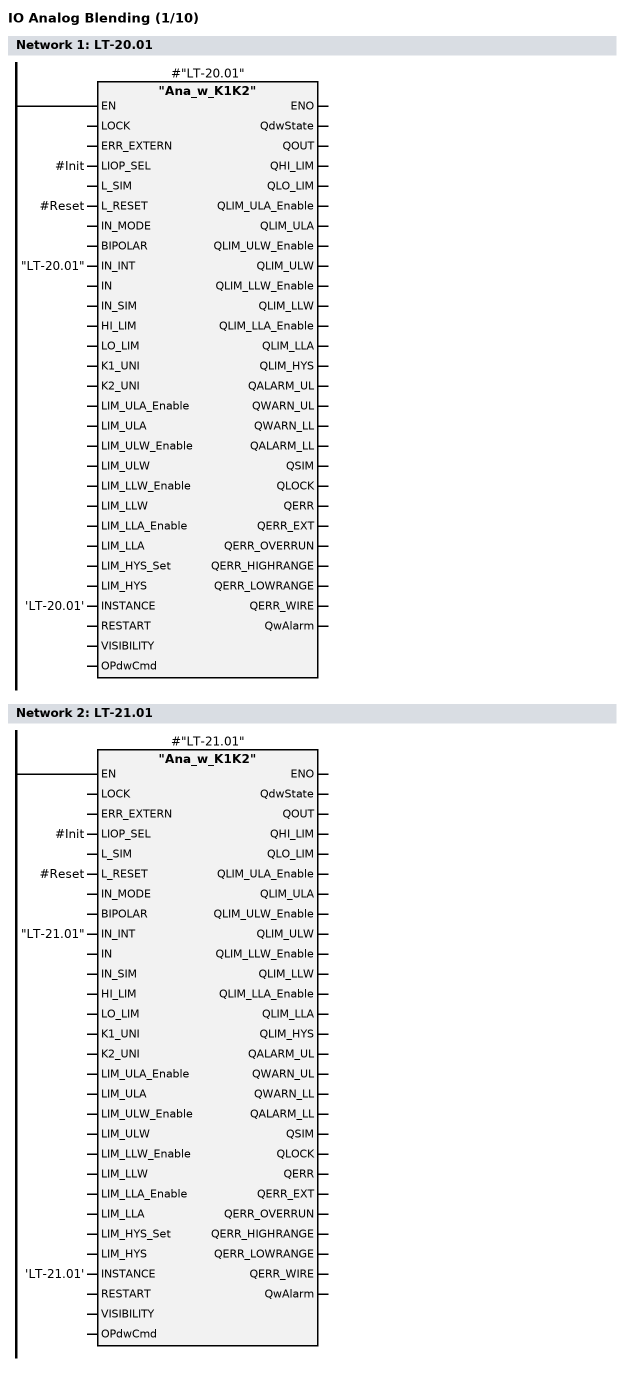
   RUNG wire#powerrail
      #"LT-20.01"(LOCK :=, ERR_EXTERN :=, LIOP_SEL := #Init, L_SIM :=, L_RESET := #Reset, IN_MODE :=, BIPOLAR :=, IN_INT := "LT-20.01", IN :=, IN_SIM :=, HI_LIM :=, LO_LIM :=, K1_UNI :=, K2_UNI :=, LIM_ULA_Enable :=, LIM_ULA :=, LIM_ULW_Enable :=, LIM_ULW :=, LIM_LLW_Enable :=, LIM_LLW :=, LIM_LLA_Enable :=, LIM_LLA :=, LIM_HYS_Set :=, LIM_HYS :=, INSTANCE := 'LT-20.01', RESTART :=, VISIBILITY :=, OPdwCmd :=, QdwState =>, QOUT =>, QHI_LIM =>, QLO_LIM =>, QLIM_ULA_Enable =>, QLIM_ULA =>, QLIM_ULW_Enable =>, QLIM_ULW =>, QLIM_LLW_Enable =>, QLIM_LLW =>, QLIM_LLA_Enable =>, QLIM_LLA =>, QLIM_HYS =>, QALARM_UL =>, QWARN_UL =>, QWARN_LL =>, QALARM_LL =>, QSIM =>, QLOCK =>, QERR =>, QERR_EXT =>, QERR_OVERRUN =>, QERR_HIGHRANGE =>, QERR_LOWRANGE =>, QERR_WIRE =>, QwAlarm =>)
   END_RUNG
   // the same network as SCL:
   #"LT-20.01"(LIOP_SEL := #Init, L_RESET := #Reset, IN_INT := "LT-20.01", INSTANCE := 'LT-20.01');   // "Ana_w_K1K2"
END_REGION

REGION Network 2: LT-21.01
   RUNG wire#powerrail
      #"LT-21.01"(LOCK :=, ERR_EXTERN :=, LIOP_SEL := #Init, L_SIM :=, L_RESET := #Reset, IN_MODE :=, BIPOLAR :=, IN_INT := "LT-21.01", IN :=, IN_SIM :=, HI_LIM :=, LO_LIM :=, K1_UNI :=, K2_UNI :=, LIM_ULA_Enable :=, LIM_ULA :=, LIM_ULW_Enable :=, LIM_ULW :=, LIM_LLW_Enable :=, LIM_LLW :=, LIM_LLA_Enable :=, LIM_LLA :=, LIM_HYS_Set :=, LIM_HYS :=, INSTANCE := 'LT-21.01', RESTART :=, VISIBILITY :=, OPdwCmd :=, QdwState =>, QOUT =>, QHI_LIM =>, QLO_LIM =>, QLIM_ULA_Enable =>, QLIM_ULA =>, QLIM_ULW_Enable =>, QLIM_ULW =>, QLIM_LLW_Enable =>, QLIM_LLW =>, QLIM_LLA_Enable =>, QLIM_LLA =>, QLIM_HYS =>, QALARM_UL =>, QWARN_UL =>, QWARN_LL =>, QALARM_LL =>, QSIM =>, QLOCK =>, QERR =>, QERR_EXT =>, QERR_OVERRUN =>, QERR_HIGHRANGE =>, QERR_LOWRANGE =>, QERR_WIRE =>, QwAlarm =>)
   END_RUNG
   // the same network as SCL:
   #"LT-21.01"(LIOP_SEL := #Init, L_RESET := #Reset, IN_INT := "LT-21.01", INSTANCE := 'LT-21.01');   // "Ana_w_K1K2"
END_REGION

REGION Network 3: LT-22.01
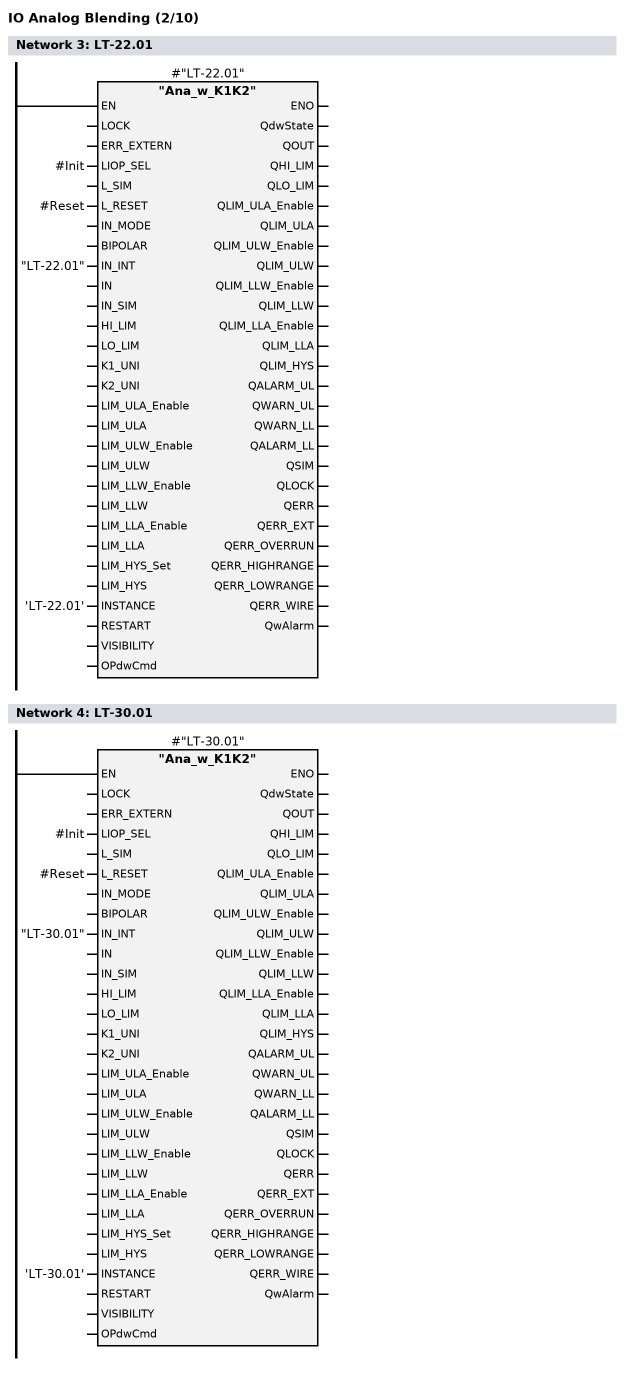
   RUNG wire#powerrail
      #"LT-22.01"(LOCK :=, ERR_EXTERN :=, LIOP_SEL := #Init, L_SIM :=, L_RESET := #Reset, IN_MODE :=, BIPOLAR :=, IN_INT := "LT-22.01", IN :=, IN_SIM :=, HI_LIM :=, LO_LIM :=, K1_UNI :=, K2_UNI :=, LIM_ULA_Enable :=, LIM_ULA :=, LIM_ULW_Enable :=, LIM_ULW :=, LIM_LLW_Enable :=, LIM_LLW :=, LIM_LLA_Enable :=, LIM_LLA :=, LIM_HYS_Set :=, LIM_HYS :=, INSTANCE := 'LT-22.01', RESTART :=, VISIBILITY :=, OPdwCmd :=, QdwState =>, QOUT =>, QHI_LIM =>, QLO_LIM =>, QLIM_ULA_Enable =>, QLIM_ULA =>, QLIM_ULW_Enable =>, QLIM_ULW =>, QLIM_LLW_Enable =>, QLIM_LLW =>, QLIM_LLA_Enable =>, QLIM_LLA =>, QLIM_HYS =>, QALARM_UL =>, QWARN_UL =>, QWARN_LL =>, QALARM_LL =>, QSIM =>, QLOCK =>, QERR =>, QERR_EXT =>, QERR_OVERRUN =>, QERR_HIGHRANGE =>, QERR_LOWRANGE =>, QERR_WIRE =>, QwAlarm =>)
   END_RUNG
   // the same network as SCL:
   #"LT-22.01"(LIOP_SEL := #Init, L_RESET := #Reset, IN_INT := "LT-22.01", INSTANCE := 'LT-22.01');   // "Ana_w_K1K2"
END_REGION

REGION Network 4: LT-30.01
   RUNG wire#powerrail
      #"LT-30.01"(LOCK :=, ERR_EXTERN :=, LIOP_SEL := #Init, L_SIM :=, L_RESET := #Reset, IN_MODE :=, BIPOLAR :=, IN_INT := "LT-30.01", IN :=, IN_SIM :=, HI_LIM :=, LO_LIM :=, K1_UNI :=, K2_UNI :=, LIM_ULA_Enable :=, LIM_ULA :=, LIM_ULW_Enable :=, LIM_ULW :=, LIM_LLW_Enable :=, LIM_LLW :=, LIM_LLA_Enable :=, LIM_LLA :=, LIM_HYS_Set :=, LIM_HYS :=, INSTANCE := 'LT-30.01', RESTART :=, VISIBILITY :=, OPdwCmd :=, QdwState =>, QOUT =>, QHI_LIM =>, QLO_LIM =>, QLIM_ULA_Enable =>, QLIM_ULA =>, QLIM_ULW_Enable =>, QLIM_ULW =>, QLIM_LLW_Enable =>, QLIM_LLW =>, QLIM_LLA_Enable =>, QLIM_LLA =>, QLIM_HYS =>, QALARM_UL =>, QWARN_UL =>, QWARN_LL =>, QALARM_LL =>, QSIM =>, QLOCK =>, QERR =>, QERR_EXT =>, QERR_OVERRUN =>, QERR_HIGHRANGE =>, QERR_LOWRANGE =>, QERR_WIRE =>, QwAlarm =>)
   END_RUNG
   // the same network as SCL:
   #"LT-30.01"(LIOP_SEL := #Init, L_RESET := #Reset, IN_INT := "LT-30.01", INSTANCE := 'LT-30.01');   // "Ana_w_K1K2"
END_REGION

REGION Network 5: LT-31.01
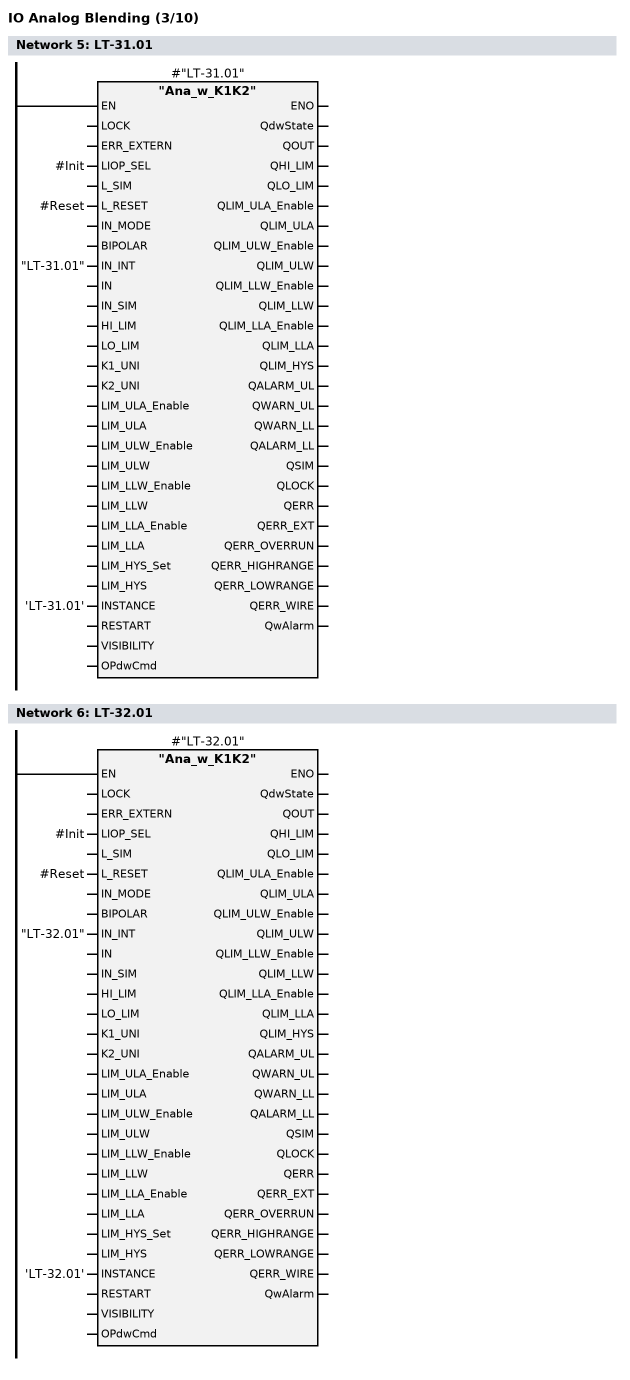
   RUNG wire#powerrail
      #"LT-31.01"(LOCK :=, ERR_EXTERN :=, LIOP_SEL := #Init, L_SIM :=, L_RESET := #Reset, IN_MODE :=, BIPOLAR :=, IN_INT := "LT-31.01", IN :=, IN_SIM :=, HI_LIM :=, LO_LIM :=, K1_UNI :=, K2_UNI :=, LIM_ULA_Enable :=, LIM_ULA :=, LIM_ULW_Enable :=, LIM_ULW :=, LIM_LLW_Enable :=, LIM_LLW :=, LIM_LLA_Enable :=, LIM_LLA :=, LIM_HYS_Set :=, LIM_HYS :=, INSTANCE := 'LT-31.01', RESTART :=, VISIBILITY :=, OPdwCmd :=, QdwState =>, QOUT =>, QHI_LIM =>, QLO_LIM =>, QLIM_ULA_Enable =>, QLIM_ULA =>, QLIM_ULW_Enable =>, QLIM_ULW =>, QLIM_LLW_Enable =>, QLIM_LLW =>, QLIM_LLA_Enable =>, QLIM_LLA =>, QLIM_HYS =>, QALARM_UL =>, QWARN_UL =>, QWARN_LL =>, QALARM_LL =>, QSIM =>, QLOCK =>, QERR =>, QERR_EXT =>, QERR_OVERRUN =>, QERR_HIGHRANGE =>, QERR_LOWRANGE =>, QERR_WIRE =>, QwAlarm =>)
   END_RUNG
   // the same network as SCL:
   #"LT-31.01"(LIOP_SEL := #Init, L_RESET := #Reset, IN_INT := "LT-31.01", INSTANCE := 'LT-31.01');   // "Ana_w_K1K2"
END_REGION

REGION Network 6: LT-32.01
   RUNG wire#powerrail
      #"LT-32.01"(LOCK :=, ERR_EXTERN :=, LIOP_SEL := #Init, L_SIM :=, L_RESET := #Reset, IN_MODE :=, BIPOLAR :=, IN_INT := "LT-32.01", IN :=, IN_SIM :=, HI_LIM :=, LO_LIM :=, K1_UNI :=, K2_UNI :=, LIM_ULA_Enable :=, LIM_ULA :=, LIM_ULW_Enable :=, LIM_ULW :=, LIM_LLW_Enable :=, LIM_LLW :=, LIM_LLA_Enable :=, LIM_LLA :=, LIM_HYS_Set :=, LIM_HYS :=, INSTANCE := 'LT-32.01', RESTART :=, VISIBILITY :=, OPdwCmd :=, QdwState =>, QOUT =>, QHI_LIM =>, QLO_LIM =>, QLIM_ULA_Enable =>, QLIM_ULA =>, QLIM_ULW_Enable =>, QLIM_ULW =>, QLIM_LLW_Enable =>, QLIM_LLW =>, QLIM_LLA_Enable =>, QLIM_LLA =>, QLIM_HYS =>, QALARM_UL =>, QWARN_UL =>, QWARN_LL =>, QALARM_LL =>, QSIM =>, QLOCK =>, QERR =>, QERR_EXT =>, QERR_OVERRUN =>, QERR_HIGHRANGE =>, QERR_LOWRANGE =>, QERR_WIRE =>, QwAlarm =>)
   END_RUNG
   // the same network as SCL:
   #"LT-32.01"(LIOP_SEL := #Init, L_RESET := #Reset, IN_INT := "LT-32.01", INSTANCE := 'LT-32.01');   // "Ana_w_K1K2"
END_REGION

REGION Network 7: LT-40.01
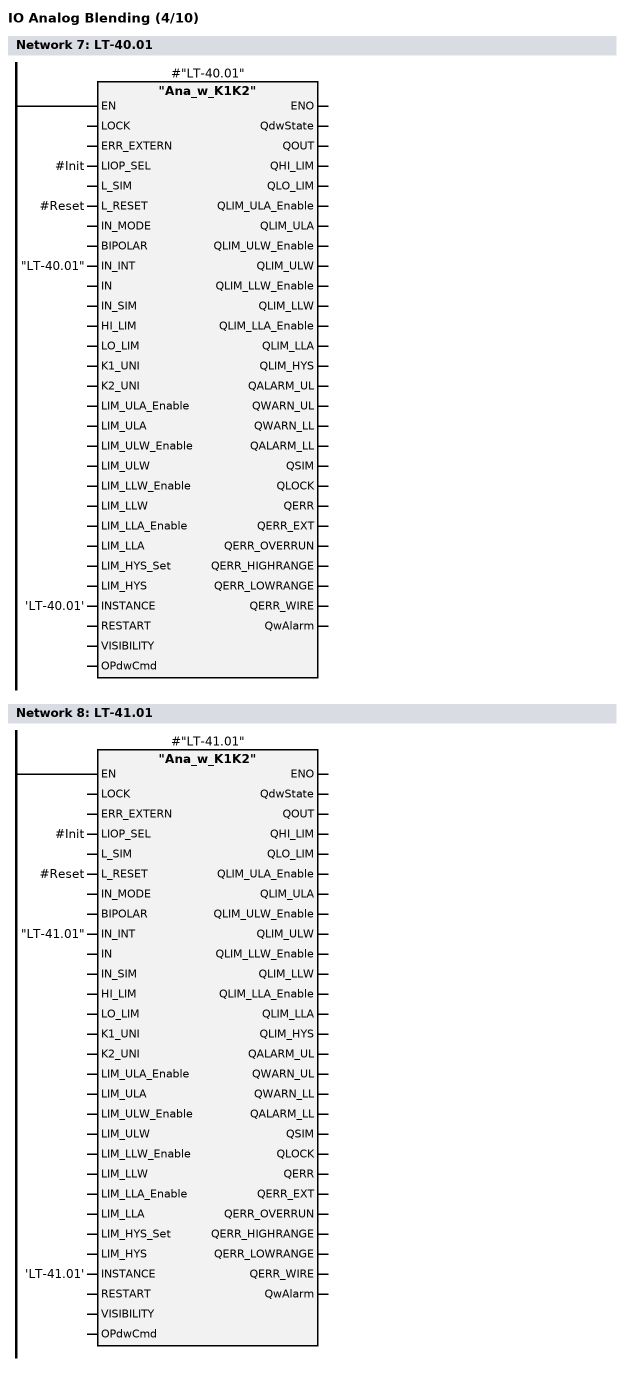
   RUNG wire#powerrail
      #"LT-40.01"(LOCK :=, ERR_EXTERN :=, LIOP_SEL := #Init, L_SIM :=, L_RESET := #Reset, IN_MODE :=, BIPOLAR :=, IN_INT := "LT-40.01", IN :=, IN_SIM :=, HI_LIM :=, LO_LIM :=, K1_UNI :=, K2_UNI :=, LIM_ULA_Enable :=, LIM_ULA :=, LIM_ULW_Enable :=, LIM_ULW :=, LIM_LLW_Enable :=, LIM_LLW :=, LIM_LLA_Enable :=, LIM_LLA :=, LIM_HYS_Set :=, LIM_HYS :=, INSTANCE := 'LT-40.01', RESTART :=, VISIBILITY :=, OPdwCmd :=, QdwState =>, QOUT =>, QHI_LIM =>, QLO_LIM =>, QLIM_ULA_Enable =>, QLIM_ULA =>, QLIM_ULW_Enable =>, QLIM_ULW =>, QLIM_LLW_Enable =>, QLIM_LLW =>, QLIM_LLA_Enable =>, QLIM_LLA =>, QLIM_HYS =>, QALARM_UL =>, QWARN_UL =>, QWARN_LL =>, QALARM_LL =>, QSIM =>, QLOCK =>, QERR =>, QERR_EXT =>, QERR_OVERRUN =>, QERR_HIGHRANGE =>, QERR_LOWRANGE =>, QERR_WIRE =>, QwAlarm =>)
   END_RUNG
   // the same network as SCL:
   #"LT-40.01"(LIOP_SEL := #Init, L_RESET := #Reset, IN_INT := "LT-40.01", INSTANCE := 'LT-40.01');   // "Ana_w_K1K2"
END_REGION

REGION Network 8: LT-41.01
   RUNG wire#powerrail
      #"LT-41.01"(LOCK :=, ERR_EXTERN :=, LIOP_SEL := #Init, L_SIM :=, L_RESET := #Reset, IN_MODE :=, BIPOLAR :=, IN_INT := "LT-41.01", IN :=, IN_SIM :=, HI_LIM :=, LO_LIM :=, K1_UNI :=, K2_UNI :=, LIM_ULA_Enable :=, LIM_ULA :=, LIM_ULW_Enable :=, LIM_ULW :=, LIM_LLW_Enable :=, LIM_LLW :=, LIM_LLA_Enable :=, LIM_LLA :=, LIM_HYS_Set :=, LIM_HYS :=, INSTANCE := 'LT-41.01', RESTART :=, VISIBILITY :=, OPdwCmd :=, QdwState =>, QOUT =>, QHI_LIM =>, QLO_LIM =>, QLIM_ULA_Enable =>, QLIM_ULA =>, QLIM_ULW_Enable =>, QLIM_ULW =>, QLIM_LLW_Enable =>, QLIM_LLW =>, QLIM_LLA_Enable =>, QLIM_LLA =>, QLIM_HYS =>, QALARM_UL =>, QWARN_UL =>, QWARN_LL =>, QALARM_LL =>, QSIM =>, QLOCK =>, QERR =>, QERR_EXT =>, QERR_OVERRUN =>, QERR_HIGHRANGE =>, QERR_LOWRANGE =>, QERR_WIRE =>, QwAlarm =>)
   END_RUNG
   // the same network as SCL:
   #"LT-41.01"(LIOP_SEL := #Init, L_RESET := #Reset, IN_INT := "LT-41.01", INSTANCE := 'LT-41.01');   // "Ana_w_K1K2"
END_REGION

REGION Network 9: FT-15.01 Communication
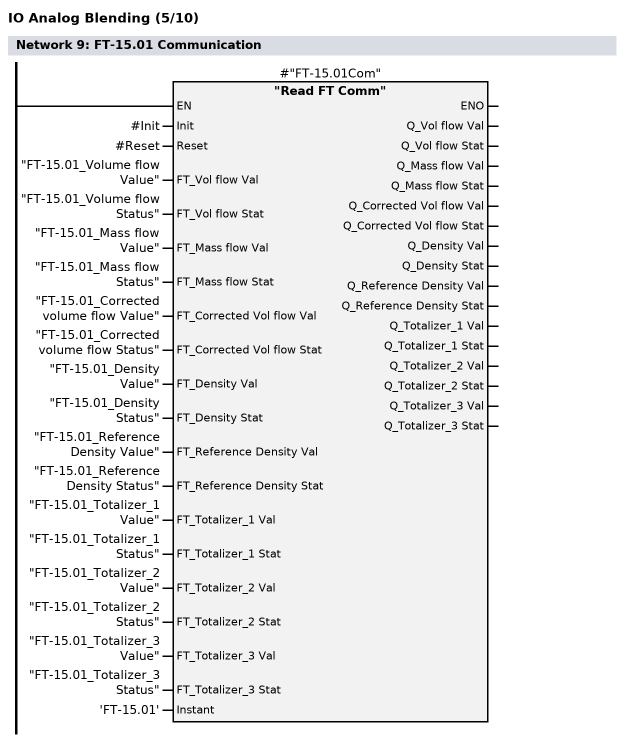
   RUNG wire#powerrail
      #"FT-15.01Com"(Init := #Init, Reset := #Reset, "FT_Vol flow Val" := "FT-15.01_Volume flow Value", "FT_Vol flow Stat" := "FT-15.01_Volume flow Status", "FT_Mass flow Val" := "FT-15.01_Mass flow Value", "FT_Mass flow Stat" := "FT-15.01_Mass flow Status", "FT_Corrected Vol flow Val" := "FT-15.01_Corrected volume flow Value", "FT_Corrected Vol flow Stat" := "FT-15.01_Corrected volume flow Status", "FT_Density Val" := "FT-15.01_Density Value", "FT_Density Stat" := "FT-15.01_Density Status", "FT_Reference Density Val" := "FT-15.01_Reference Density Value", "FT_Reference Density Stat" := "FT-15.01_Reference Density Status", "FT_Totalizer_1 Val" := "FT-15.01_Totalizer_1 Value", "FT_Totalizer_1 Stat" := "FT-15.01_Totalizer_1 Status", "FT_Totalizer_2 Val" := "FT-15.01_Totalizer_2 Value", "FT_Totalizer_2 Stat" := "FT-15.01_Totalizer_2 Status", "FT_Totalizer_3 Val" := "FT-15.01_Totalizer_3 Value", "FT_Totalizer_3 Stat" := "FT-15.01_Totalizer_3 Status", Instant := 'FT-15.01', "Q_Vol flow Val" =>, "Q_Vol flow Stat" =>, "Q_Mass flow Val" =>, "Q_Mass flow Stat" =>, "Q_Corrected Vol flow Val" =>, "Q_Corrected Vol flow Stat" =>, "Q_Density Val" =>, "Q_Density Stat" =>, "Q_Reference Density Val" =>, "Q_Reference Density Stat" =>, "Q_Totalizer_1 Val" =>, "Q_Totalizer_1 Stat" =>, "Q_Totalizer_2 Val" =>, "Q_Totalizer_2 Stat" =>, "Q_Totalizer_3 Val" =>, "Q_Totalizer_3 Stat" =>)
   END_RUNG
   // the same network as SCL:
   #"FT-15.01Com"(Init := #Init,   // "Read FT Comm"
                  Reset := #Reset,
                  "FT_Vol flow Val" := "FT-15.01_Volume flow Value",
                  "FT_Vol flow Stat" := "FT-15.01_Volume flow Status",
                  "FT_Mass flow Val" := "FT-15.01_Mass flow Value",
                  "FT_Mass flow Stat" := "FT-15.01_Mass flow Status",
                  "FT_Corrected Vol flow Val" := "FT-15.01_Corrected volume flow Value",
                  "FT_Corrected Vol flow Stat" := "FT-15.01_Corrected volume flow Status",
                  "FT_Density Val" := "FT-15.01_Density Value",
                  "FT_Density Stat" := "FT-15.01_Density Status",
                  "FT_Reference Density Val" := "FT-15.01_Reference Density Value",
                  "FT_Reference Density Stat" := "FT-15.01_Reference Density Status",
                  "FT_Totalizer_1 Val" := "FT-15.01_Totalizer_1 Value",
                  "FT_Totalizer_1 Stat" := "FT-15.01_Totalizer_1 Status",
                  "FT_Totalizer_2 Val" := "FT-15.01_Totalizer_2 Value",
                  "FT_Totalizer_2 Stat" := "FT-15.01_Totalizer_2 Status",
                  "FT_Totalizer_3 Val" := "FT-15.01_Totalizer_3 Value",
                  "FT_Totalizer_3 Stat" := "FT-15.01_Totalizer_3 Status",
                  Instant := 'FT-15.01');
END_REGION

REGION Network 10: FT-15.01 Flowrate
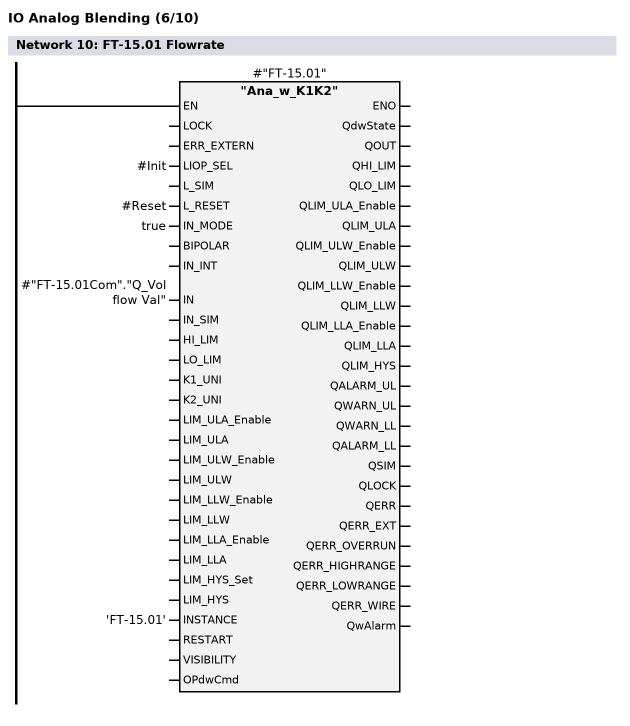
   RUNG wire#powerrail
      #"FT-15.01"(LOCK :=, ERR_EXTERN :=, LIOP_SEL := #Init, L_SIM :=, L_RESET := #Reset, IN_MODE := true, BIPOLAR :=, IN_INT :=, IN := #"FT-15.01Com"."Q_Vol flow Val", IN_SIM :=, HI_LIM :=, LO_LIM :=, K1_UNI :=, K2_UNI :=, LIM_ULA_Enable :=, LIM_ULA :=, LIM_ULW_Enable :=, LIM_ULW :=, LIM_LLW_Enable :=, LIM_LLW :=, LIM_LLA_Enable :=, LIM_LLA :=, LIM_HYS_Set :=, LIM_HYS :=, INSTANCE := 'FT-15.01', RESTART :=, VISIBILITY :=, OPdwCmd :=, QdwState =>, QOUT =>, QHI_LIM =>, QLO_LIM =>, QLIM_ULA_Enable =>, QLIM_ULA =>, QLIM_ULW_Enable =>, QLIM_ULW =>, QLIM_LLW_Enable =>, QLIM_LLW =>, QLIM_LLA_Enable =>, QLIM_LLA =>, QLIM_HYS =>, QALARM_UL =>, QWARN_UL =>, QWARN_LL =>, QALARM_LL =>, QSIM =>, QLOCK =>, QERR =>, QERR_EXT =>, QERR_OVERRUN =>, QERR_HIGHRANGE =>, QERR_LOWRANGE =>, QERR_WIRE =>, QwAlarm =>)
   END_RUNG
   // the same network as SCL:
   #"FT-15.01"(LIOP_SEL := #Init,   // "Ana_w_K1K2"
               L_RESET := #Reset,
               IN_MODE := true,
               IN := #"FT-15.01Com"."Q_Vol flow Val",
               INSTANCE := 'FT-15.01');
END_REGION

REGION Network 11: FT-22.01 Communication
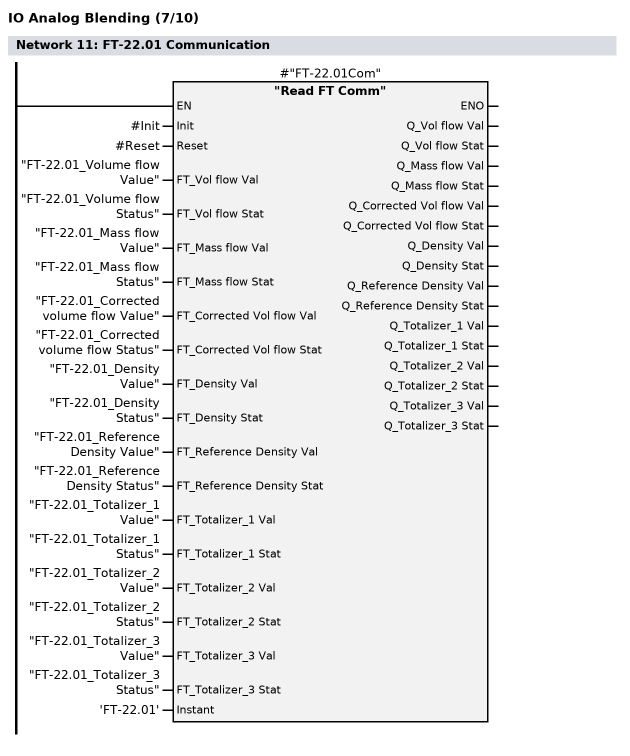
   RUNG wire#powerrail
      #"FT-22.01Com"(Init := #Init, Reset := #Reset, "FT_Vol flow Val" := "FT-22.01_Volume flow Value", "FT_Vol flow Stat" := "FT-22.01_Volume flow Status", "FT_Mass flow Val" := "FT-22.01_Mass flow Value", "FT_Mass flow Stat" := "FT-22.01_Mass flow Status", "FT_Corrected Vol flow Val" := "FT-22.01_Corrected volume flow Value", "FT_Corrected Vol flow Stat" := "FT-22.01_Corrected volume flow Status", "FT_Density Val" := "FT-22.01_Density Value", "FT_Density Stat" := "FT-22.01_Density Status", "FT_Reference Density Val" := "FT-22.01_Reference Density Value", "FT_Reference Density Stat" := "FT-22.01_Reference Density Status", "FT_Totalizer_1 Val" := "FT-22.01_Totalizer_1 Value", "FT_Totalizer_1 Stat" := "FT-22.01_Totalizer_1 Status", "FT_Totalizer_2 Val" := "FT-22.01_Totalizer_2 Value", "FT_Totalizer_2 Stat" := "FT-22.01_Totalizer_2 Status", "FT_Totalizer_3 Val" := "FT-22.01_Totalizer_3 Value", "FT_Totalizer_3 Stat" := "FT-22.01_Totalizer_3 Status", Instant := 'FT-22.01', "Q_Vol flow Val" =>, "Q_Vol flow Stat" =>, "Q_Mass flow Val" =>, "Q_Mass flow Stat" =>, "Q_Corrected Vol flow Val" =>, "Q_Corrected Vol flow Stat" =>, "Q_Density Val" =>, "Q_Density Stat" =>, "Q_Reference Density Val" =>, "Q_Reference Density Stat" =>, "Q_Totalizer_1 Val" =>, "Q_Totalizer_1 Stat" =>, "Q_Totalizer_2 Val" =>, "Q_Totalizer_2 Stat" =>, "Q_Totalizer_3 Val" =>, "Q_Totalizer_3 Stat" =>)
   END_RUNG
   // the same network as SCL:
   #"FT-22.01Com"(Init := #Init,   // "Read FT Comm"
                  Reset := #Reset,
                  "FT_Vol flow Val" := "FT-22.01_Volume flow Value",
                  "FT_Vol flow Stat" := "FT-22.01_Volume flow Status",
                  "FT_Mass flow Val" := "FT-22.01_Mass flow Value",
                  "FT_Mass flow Stat" := "FT-22.01_Mass flow Status",
                  "FT_Corrected Vol flow Val" := "FT-22.01_Corrected volume flow Value",
                  "FT_Corrected Vol flow Stat" := "FT-22.01_Corrected volume flow Status",
                  "FT_Density Val" := "FT-22.01_Density Value",
                  "FT_Density Stat" := "FT-22.01_Density Status",
                  "FT_Reference Density Val" := "FT-22.01_Reference Density Value",
                  "FT_Reference Density Stat" := "FT-22.01_Reference Density Status",
                  "FT_Totalizer_1 Val" := "FT-22.01_Totalizer_1 Value",
                  "FT_Totalizer_1 Stat" := "FT-22.01_Totalizer_1 Status",
                  "FT_Totalizer_2 Val" := "FT-22.01_Totalizer_2 Value",
                  "FT_Totalizer_2 Stat" := "FT-22.01_Totalizer_2 Status",
                  "FT_Totalizer_3 Val" := "FT-22.01_Totalizer_3 Value",
                  "FT_Totalizer_3 Stat" := "FT-22.01_Totalizer_3 Status",
                  Instant := 'FT-22.01');
END_REGION

REGION Network 12: FT-22.01 Flowrate
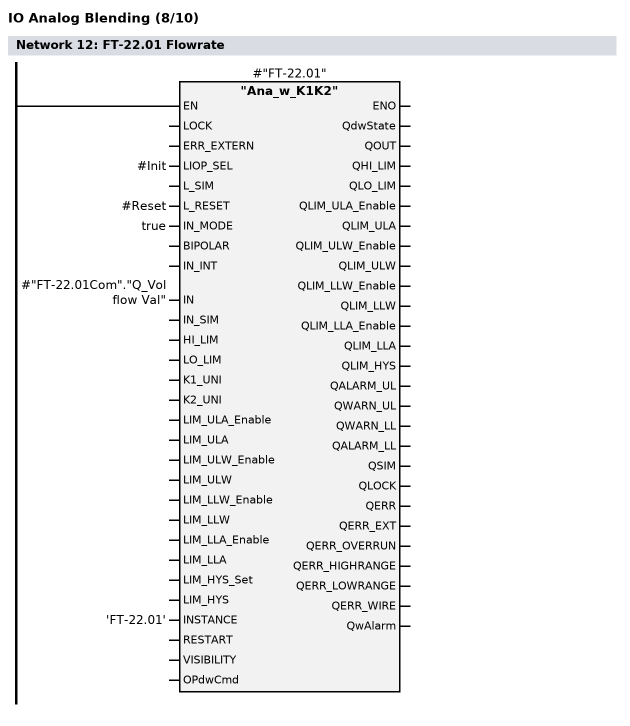
   RUNG wire#powerrail
      #"FT-22.01"(LOCK :=, ERR_EXTERN :=, LIOP_SEL := #Init, L_SIM :=, L_RESET := #Reset, IN_MODE := true, BIPOLAR :=, IN_INT :=, IN := #"FT-22.01Com"."Q_Vol flow Val", IN_SIM :=, HI_LIM :=, LO_LIM :=, K1_UNI :=, K2_UNI :=, LIM_ULA_Enable :=, LIM_ULA :=, LIM_ULW_Enable :=, LIM_ULW :=, LIM_LLW_Enable :=, LIM_LLW :=, LIM_LLA_Enable :=, LIM_LLA :=, LIM_HYS_Set :=, LIM_HYS :=, INSTANCE := 'FT-22.01', RESTART :=, VISIBILITY :=, OPdwCmd :=, QdwState =>, QOUT =>, QHI_LIM =>, QLO_LIM =>, QLIM_ULA_Enable =>, QLIM_ULA =>, QLIM_ULW_Enable =>, QLIM_ULW =>, QLIM_LLW_Enable =>, QLIM_LLW =>, QLIM_LLA_Enable =>, QLIM_LLA =>, QLIM_HYS =>, QALARM_UL =>, QWARN_UL =>, QWARN_LL =>, QALARM_LL =>, QSIM =>, QLOCK =>, QERR =>, QERR_EXT =>, QERR_OVERRUN =>, QERR_HIGHRANGE =>, QERR_LOWRANGE =>, QERR_WIRE =>, QwAlarm =>)
   END_RUNG
   // the same network as SCL:
   #"FT-22.01"(LIOP_SEL := #Init,   // "Ana_w_K1K2"
               L_RESET := #Reset,
               IN_MODE := true,
               IN := #"FT-22.01Com"."Q_Vol flow Val",
               INSTANCE := 'FT-22.01');
END_REGION

REGION Network 13: FT-32.01 Communication
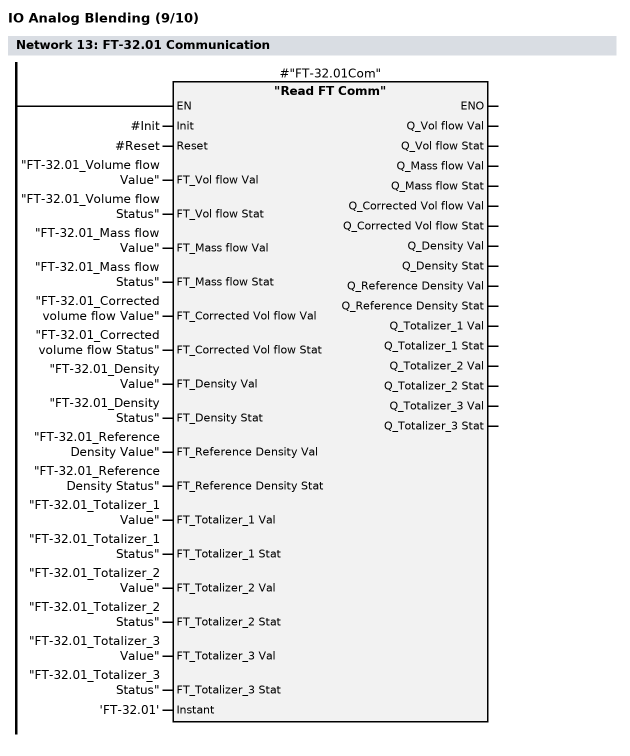
   RUNG wire#powerrail
      #"FT-32.01Com"(Init := #Init, Reset := #Reset, "FT_Vol flow Val" := "FT-32.01_Volume flow Value", "FT_Vol flow Stat" := "FT-32.01_Volume flow Status", "FT_Mass flow Val" := "FT-32.01_Mass flow Value", "FT_Mass flow Stat" := "FT-32.01_Mass flow Status", "FT_Corrected Vol flow Val" := "FT-32.01_Corrected volume flow Value", "FT_Corrected Vol flow Stat" := "FT-32.01_Corrected volume flow Status", "FT_Density Val" := "FT-32.01_Density Value", "FT_Density Stat" := "FT-32.01_Density Status", "FT_Reference Density Val" := "FT-32.01_Reference Density Value", "FT_Reference Density Stat" := "FT-32.01_Reference Density Status", "FT_Totalizer_1 Val" := "FT-32.01_Totalizer_1 Value", "FT_Totalizer_1 Stat" := "FT-32.01_Totalizer_1 Status", "FT_Totalizer_2 Val" := "FT-32.01_Totalizer_2 Value", "FT_Totalizer_2 Stat" := "FT-32.01_Totalizer_2 Status", "FT_Totalizer_3 Val" := "FT-32.01_Totalizer_3 Value", "FT_Totalizer_3 Stat" := "FT-32.01_Totalizer_3 Status", Instant := 'FT-32.01', "Q_Vol flow Val" =>, "Q_Vol flow Stat" =>, "Q_Mass flow Val" =>, "Q_Mass flow Stat" =>, "Q_Corrected Vol flow Val" =>, "Q_Corrected Vol flow Stat" =>, "Q_Density Val" =>, "Q_Density Stat" =>, "Q_Reference Density Val" =>, "Q_Reference Density Stat" =>, "Q_Totalizer_1 Val" =>, "Q_Totalizer_1 Stat" =>, "Q_Totalizer_2 Val" =>, "Q_Totalizer_2 Stat" =>, "Q_Totalizer_3 Val" =>, "Q_Totalizer_3 Stat" =>)
   END_RUNG
   // the same network as SCL:
   #"FT-32.01Com"(Init := #Init,   // "Read FT Comm"
                  Reset := #Reset,
                  "FT_Vol flow Val" := "FT-32.01_Volume flow Value",
                  "FT_Vol flow Stat" := "FT-32.01_Volume flow Status",
                  "FT_Mass flow Val" := "FT-32.01_Mass flow Value",
                  "FT_Mass flow Stat" := "FT-32.01_Mass flow Status",
                  "FT_Corrected Vol flow Val" := "FT-32.01_Corrected volume flow Value",
                  "FT_Corrected Vol flow Stat" := "FT-32.01_Corrected volume flow Status",
                  "FT_Density Val" := "FT-32.01_Density Value",
                  "FT_Density Stat" := "FT-32.01_Density Status",
                  "FT_Reference Density Val" := "FT-32.01_Reference Density Value",
                  "FT_Reference Density Stat" := "FT-32.01_Reference Density Status",
                  "FT_Totalizer_1 Val" := "FT-32.01_Totalizer_1 Value",
                  "FT_Totalizer_1 Stat" := "FT-32.01_Totalizer_1 Status",
                  "FT_Totalizer_2 Val" := "FT-32.01_Totalizer_2 Value",
                  "FT_Totalizer_2 Stat" := "FT-32.01_Totalizer_2 Status",
                  "FT_Totalizer_3 Val" := "FT-32.01_Totalizer_3 Value",
                  "FT_Totalizer_3 Stat" := "FT-32.01_Totalizer_3 Status",
                  Instant := 'FT-32.01');
END_REGION

REGION Network 14: FT-32.01 Flowrate
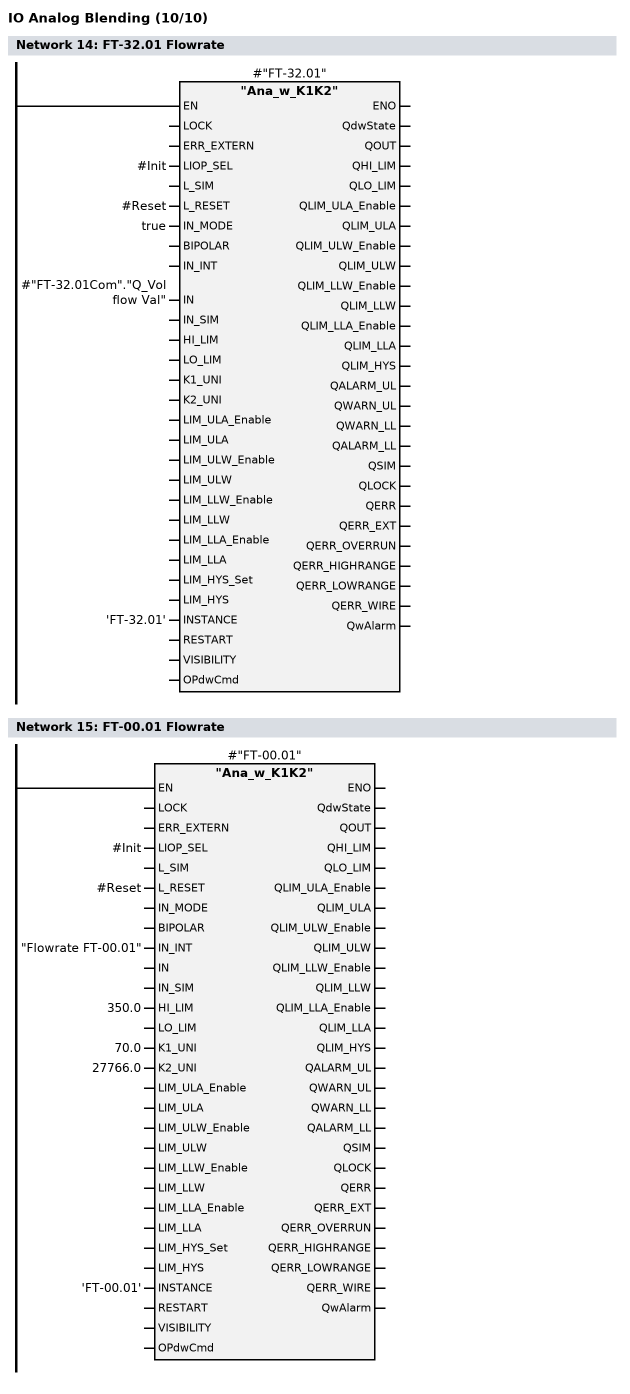
   RUNG wire#powerrail
      #"FT-32.01"(LOCK :=, ERR_EXTERN :=, LIOP_SEL := #Init, L_SIM :=, L_RESET := #Reset, IN_MODE := true, BIPOLAR :=, IN_INT :=, IN := #"FT-32.01Com"."Q_Vol flow Val", IN_SIM :=, HI_LIM :=, LO_LIM :=, K1_UNI :=, K2_UNI :=, LIM_ULA_Enable :=, LIM_ULA :=, LIM_ULW_Enable :=, LIM_ULW :=, LIM_LLW_Enable :=, LIM_LLW :=, LIM_LLA_Enable :=, LIM_LLA :=, LIM_HYS_Set :=, LIM_HYS :=, INSTANCE := 'FT-32.01', RESTART :=, VISIBILITY :=, OPdwCmd :=, QdwState =>, QOUT =>, QHI_LIM =>, QLO_LIM =>, QLIM_ULA_Enable =>, QLIM_ULA =>, QLIM_ULW_Enable =>, QLIM_ULW =>, QLIM_LLW_Enable =>, QLIM_LLW =>, QLIM_LLA_Enable =>, QLIM_LLA =>, QLIM_HYS =>, QALARM_UL =>, QWARN_UL =>, QWARN_LL =>, QALARM_LL =>, QSIM =>, QLOCK =>, QERR =>, QERR_EXT =>, QERR_OVERRUN =>, QERR_HIGHRANGE =>, QERR_LOWRANGE =>, QERR_WIRE =>, QwAlarm =>)
   END_RUNG
   // the same network as SCL:
   #"FT-32.01"(LIOP_SEL := #Init,   // "Ana_w_K1K2"
               L_RESET := #Reset,
               IN_MODE := true,
               IN := #"FT-32.01Com"."Q_Vol flow Val",
               INSTANCE := 'FT-32.01');
END_REGION

REGION Network 15: FT-00.01 Flowrate
   RUNG wire#powerrail
      #"FT-00.01"(LOCK :=, ERR_EXTERN :=, LIOP_SEL := #Init, L_SIM :=, L_RESET := #Reset, IN_MODE :=, BIPOLAR :=, IN_INT := "Flowrate FT-00.01", IN :=, IN_SIM :=, HI_LIM := 350.0, LO_LIM :=, K1_UNI := 70.0, K2_UNI := 27766.0, LIM_ULA_Enable :=, LIM_ULA :=, LIM_ULW_Enable :=, LIM_ULW :=, LIM_LLW_Enable :=, LIM_LLW :=, LIM_LLA_Enable :=, LIM_LLA :=, LIM_HYS_Set :=, LIM_HYS :=, INSTANCE := 'FT-00.01', RESTART :=, VISIBILITY :=, OPdwCmd :=, QdwState =>, QOUT =>, QHI_LIM =>, QLO_LIM =>, QLIM_ULA_Enable =>, QLIM_ULA =>, QLIM_ULW_Enable =>, QLIM_ULW =>, QLIM_LLW_Enable =>, QLIM_LLW =>, QLIM_LLA_Enable =>, QLIM_LLA =>, QLIM_HYS =>, QALARM_UL =>, QWARN_UL =>, QWARN_LL =>, QALARM_LL =>, QSIM =>, QLOCK =>, QERR =>, QERR_EXT =>, QERR_OVERRUN =>, QERR_HIGHRANGE =>, QERR_LOWRANGE =>, QERR_WIRE =>, QwAlarm =>)
   END_RUNG
   // the same network as SCL:
   #"FT-00.01"(LIOP_SEL := #Init,   // "Ana_w_K1K2"
               L_RESET := #Reset,
               IN_INT := "Flowrate FT-00.01",
               HI_LIM := 350.0,
               K1_UNI := 70.0,
               K2_UNI := 27766.0,
               INSTANCE := 'FT-00.01');
END_REGION
END_FUNCTION_BLOCK

FUNCTION_BLOCK "IO Digital Blending"   // FB6, LAD
{ S7_Optimized_Access := 'FALSE' }
VERSION : 0.1
// stored: AutoNumber true, IsIECCheckEnabled false, SetENOAutomatically false, UDAEnableTagReadback false
   VAR_INPUT
      Init : Bool;
      Reset : Bool;
   END_VAR
   VAR
      "DRP-P22.01" { S7_SetPoint := 'True'} : "Digital";   // DRY RUN PROTECTION MONO PUMP P-22.01
      "DRP-P32.01" { S7_SetPoint := 'True'} : "Digital";   // DRY RUN PROTECTION MONO PUMP P-32.01
   END_VAR
BEGIN

REGION Network 1: DRP-P22.01
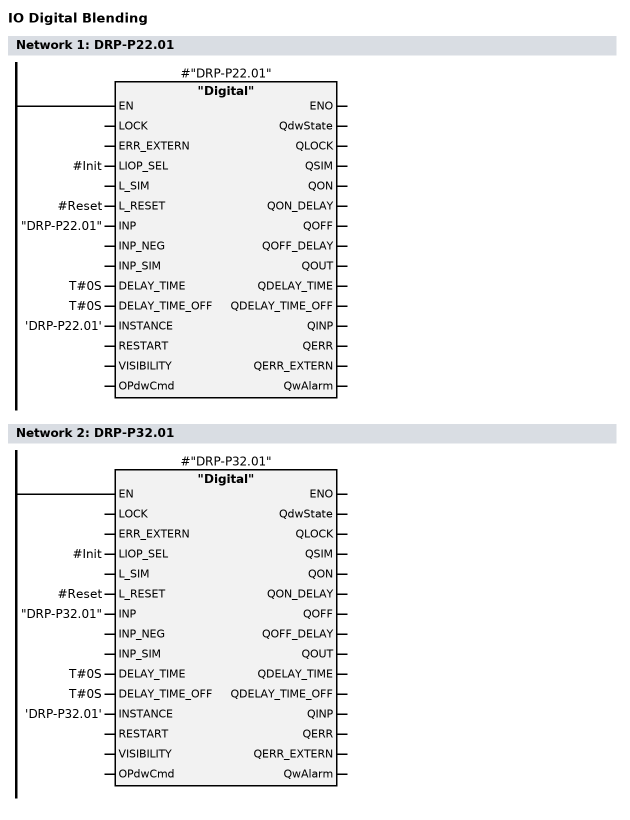
   RUNG wire#powerrail
      #"DRP-P22.01"(LOCK :=, ERR_EXTERN :=, LIOP_SEL := #Init, L_SIM :=, L_RESET := #Reset, INP := "DRP-P22.01", INP_NEG :=, INP_SIM :=, DELAY_TIME := T#0S, DELAY_TIME_OFF := T#0S, INSTANCE := 'DRP-P22.01', RESTART :=, VISIBILITY :=, OPdwCmd :=, QdwState =>, QLOCK =>, QSIM =>, QON =>, QON_DELAY =>, QOFF =>, QOFF_DELAY =>, QOUT =>, QDELAY_TIME =>, QDELAY_TIME_OFF =>, QINP =>, QERR =>, QERR_EXTERN =>, QwAlarm =>)
   END_RUNG
   // the same network as SCL:
   #"DRP-P22.01"(LIOP_SEL := #Init,   // "Digital"
                 L_RESET := #Reset,
                 INP := "DRP-P22.01",
                 DELAY_TIME := T#0S,
                 DELAY_TIME_OFF := T#0S,
                 INSTANCE := 'DRP-P22.01');
END_REGION

REGION Network 2: DRP-P32.01
   RUNG wire#powerrail
      #"DRP-P32.01"(LOCK :=, ERR_EXTERN :=, LIOP_SEL := #Init, L_SIM :=, L_RESET := #Reset, INP := "DRP-P32.01", INP_NEG :=, INP_SIM :=, DELAY_TIME := T#0S, DELAY_TIME_OFF := T#0S, INSTANCE := 'DRP-P32.01', RESTART :=, VISIBILITY :=, OPdwCmd :=, QdwState =>, QLOCK =>, QSIM =>, QON =>, QON_DELAY =>, QOFF =>, QOFF_DELAY =>, QOUT =>, QDELAY_TIME =>, QDELAY_TIME_OFF =>, QINP =>, QERR =>, QERR_EXTERN =>, QwAlarm =>)
   END_RUNG
   // the same network as SCL:
   #"DRP-P32.01"(LIOP_SEL := #Init,   // "Digital"
                 L_RESET := #Reset,
                 INP := "DRP-P32.01",
                 DELAY_TIME := T#0S,
                 DELAY_TIME_OFF := T#0S,
                 INSTANCE := 'DRP-P32.01');
END_REGION
END_FUNCTION_BLOCK

FUNCTION_BLOCK "Alarm Flow Collector"   // FB211, LAD
{ S7_Optimized_Access := 'TRUE' }
VERSION : 0.1
// stored: AutoNumber false, IsIECCheckEnabled false, IsRetainMemResEnabled false, MemoryReserve 100, SetENOAutomatically false, UDAEnableTagReadback false
   VAR_INPUT
      Reset : Bool;
   END_VAR
   VAR
      alwaysON : Bool;
   END_VAR
   VAR RETAIN
      Param : Struct
         min_Flow : Struct
            ChiliAwetan1 : Real := 5.0;
            ChiliAwetan2 : Real := 5.0;
            ChiliAwetan3 : Real := 5.0;
            Tomato : Real := 5.0;
            ChiliFresh1 : Real := 5.0;
            ChiliFresh2 : Real := 5.0;
            ChiliFresh3 : Real := 5.0;
            Garlic : Real := 5.0;
            HW : Real := 5.0;
            Vinegar : Real := 5.0;
            Sugar : Real := 5.0;
            Salt : Real := 5.0;
            ProWater : Real := 5.0;
            Homomixer : Real := 5.0;
         END_STRUCT;
         timerMon : Struct
            ChiliAwetan1 : TON_TIME;
            ChiliAwetan2 : TON_TIME;
            ChiliAwetan3 : TON_TIME;
            Tomato : TON_TIME;
            ChiliFresh1 : TON_TIME;
            ChiliFresh2 : TON_TIME;
            ChiliFresh3 : TON_TIME;
            Garlic : TON_TIME;
            HW : TON_TIME;
            Vinegar : TON_TIME;
            Sugar : TON_TIME;
            Salt : TON_TIME;
            ProWater : TON_TIME;
            Homomixer : TON_TIME;
         END_STRUCT;
      END_STRUCT;
   END_VAR
   VAR
      AlarmFlow_Blend : Word;
   END_VAR
   // Param.timerMon.ChiliAwetan1.PT := T#20s;
   // Param.timerMon.ChiliAwetan2.PT := T#20s;
   // Param.timerMon.ChiliAwetan3.PT := T#20s;
   // Param.timerMon.Tomato.PT := T#20s;
   // Param.timerMon.ChiliFresh1.PT := T#20s;
   // Param.timerMon.ChiliFresh2.PT := T#20s;
   // Param.timerMon.ChiliFresh3.PT := T#20s;
   // Param.timerMon.Garlic.PT := T#20s;
   // Param.timerMon.HW.PT := T#20s;
   // Param.timerMon.Vinegar.PT := T#20s;
   // Param.timerMon.Sugar.PT := T#20s;
   // Param.timerMon.Salt.PT := T#20s;
   // Param.timerMon.ProWater.PT := T#20s;
   // Param.timerMon.Homomixer.PT := T#20s;
BEGIN

REGION Network 1: always ON
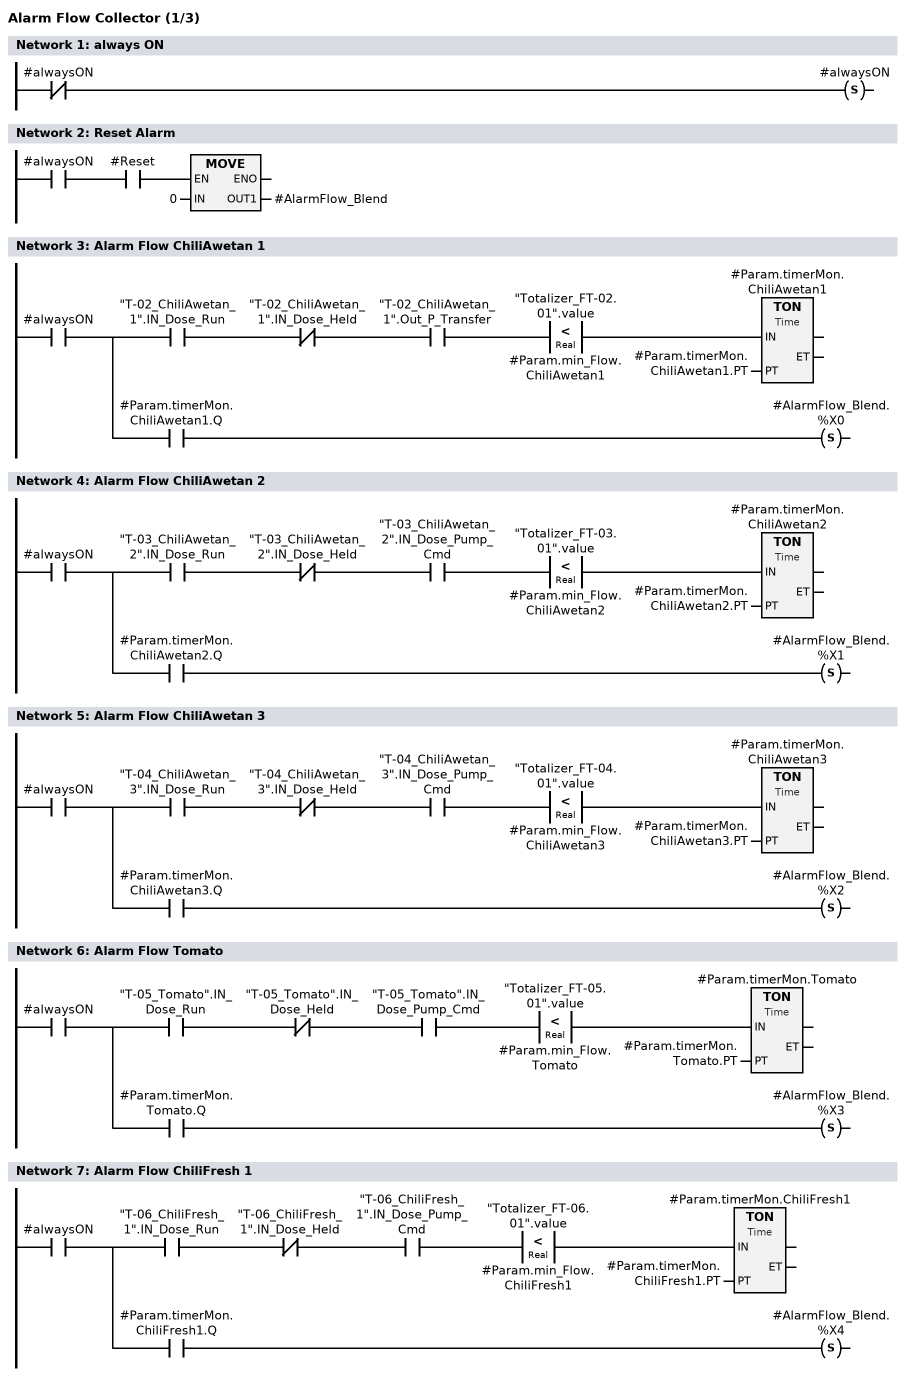
   RUNG wire#powerrail
      I_Contact( #alwaysON )
      S_Coil( #alwaysON )
   END_RUNG
   // the same network as SCL:
   IF NOT #alwaysON THEN #alwaysON := TRUE; END_IF;
END_REGION

REGION Network 2: Reset Alarm
   RUNG wire#powerrail
      Contact( #alwaysON )
      Contact( #Reset )
      Move(in := 0, out1 => #AlarmFlow_Blend)
   END_RUNG
   // the same network as SCL:
   IF #alwaysON AND #Reset THEN #AlarmFlow_Blend := 0; END_IF;
END_REGION

REGION Network 3: Alarm Flow ChiliAwetan 1
   RUNG wire#powerrail
      Contact( #alwaysON )
      wire#w1
      Contact( "T-02_ChiliAwetan_1".IN_Dose_Run )
      I_Contact( "T-02_ChiliAwetan_1".IN_Dose_Held )
      Contact( "T-02_ChiliAwetan_1".Out_P_Transfer )
      { S7_Templates := "SrcType := Real" } LT_Contact(in1 := "Totalizer_FT-02.01".value, in2 := #Param.min_Flow.ChiliAwetan1)
      { S7_Templates := "time_type := Time" } #Param.timerMon.ChiliAwetan1.TON(pt := #Param.timerMon.ChiliAwetan1.PT, et =>)
   END_RUNG
   RUNG wire#w1
      Contact( #Param.timerMon.ChiliAwetan1.Q )
      S_Coil( #AlarmFlow_Blend.%X0 )
   END_RUNG
   // the same network as SCL:
   #Param.timerMon.ChiliAwetan1.TON(IN := #alwaysON AND "T-02_ChiliAwetan_1".IN_Dose_Run AND NOT "T-02_ChiliAwetan_1".IN_Dose_Held AND "T-02_ChiliAwetan_1".Out_P_Transfer AND ("Totalizer_FT-02.01".value < #Param.min_Flow.ChiliAwetan1),
                           PT := #Param.timerMon.ChiliAwetan1.PT);
   IF #alwaysON AND #Param.timerMon.ChiliAwetan1.Q THEN #AlarmFlow_Blend.%X0 := TRUE; END_IF;
END_REGION

REGION Network 4: Alarm Flow ChiliAwetan 2
   RUNG wire#powerrail
      Contact( #alwaysON )
      wire#w1
      Contact( "T-03_ChiliAwetan_2".IN_Dose_Run )
      I_Contact( "T-03_ChiliAwetan_2".IN_Dose_Held )
      Contact( "T-03_ChiliAwetan_2".IN_Dose_Pump_Cmd )
      { S7_Templates := "SrcType := Real" } LT_Contact(in1 := "Totalizer_FT-03.01".value, in2 := #Param.min_Flow.ChiliAwetan2)
      { S7_Templates := "time_type := Time" } #Param.timerMon.ChiliAwetan2.TON(pt := #Param.timerMon.ChiliAwetan2.PT, et =>)
   END_RUNG
   RUNG wire#w1
      Contact( #Param.timerMon.ChiliAwetan2.Q )
      S_Coil( #AlarmFlow_Blend.%X1 )
   END_RUNG
   // the same network as SCL:
   #Param.timerMon.ChiliAwetan2.TON(IN := #alwaysON AND "T-03_ChiliAwetan_2".IN_Dose_Run AND NOT "T-03_ChiliAwetan_2".IN_Dose_Held AND "T-03_ChiliAwetan_2".IN_Dose_Pump_Cmd AND ("Totalizer_FT-03.01".value < #Param.min_Flow.ChiliAwetan2),
                           PT := #Param.timerMon.ChiliAwetan2.PT);
   IF #alwaysON AND #Param.timerMon.ChiliAwetan2.Q THEN #AlarmFlow_Blend.%X1 := TRUE; END_IF;
END_REGION

REGION Network 5: Alarm Flow ChiliAwetan 3
   RUNG wire#powerrail
      Contact( #alwaysON )
      wire#w1
      Contact( "T-04_ChiliAwetan_3".IN_Dose_Run )
      I_Contact( "T-04_ChiliAwetan_3".IN_Dose_Held )
      Contact( "T-04_ChiliAwetan_3".IN_Dose_Pump_Cmd )
      { S7_Templates := "SrcType := Real" } LT_Contact(in1 := "Totalizer_FT-04.01".value, in2 := #Param.min_Flow.ChiliAwetan3)
      { S7_Templates := "time_type := Time" } #Param.timerMon.ChiliAwetan3.TON(pt := #Param.timerMon.ChiliAwetan3.PT, et =>)
   END_RUNG
   RUNG wire#w1
      Contact( #Param.timerMon.ChiliAwetan3.Q )
      S_Coil( #AlarmFlow_Blend.%X2 )
   END_RUNG
   // the same network as SCL:
   #Param.timerMon.ChiliAwetan3.TON(IN := #alwaysON AND "T-04_ChiliAwetan_3".IN_Dose_Run AND NOT "T-04_ChiliAwetan_3".IN_Dose_Held AND "T-04_ChiliAwetan_3".IN_Dose_Pump_Cmd AND ("Totalizer_FT-04.01".value < #Param.min_Flow.ChiliAwetan3),
                           PT := #Param.timerMon.ChiliAwetan3.PT);
   IF #alwaysON AND #Param.timerMon.ChiliAwetan3.Q THEN #AlarmFlow_Blend.%X2 := TRUE; END_IF;
END_REGION

REGION Network 6: Alarm Flow Tomato
   RUNG wire#powerrail
      Contact( #alwaysON )
      wire#w1
      Contact( "T-05_Tomato".IN_Dose_Run )
      I_Contact( "T-05_Tomato".IN_Dose_Held )
      Contact( "T-05_Tomato".IN_Dose_Pump_Cmd )
      { S7_Templates := "SrcType := Real" } LT_Contact(in1 := "Totalizer_FT-05.01".value, in2 := #Param.min_Flow.Tomato)
      { S7_Templates := "time_type := Time" } #Param.timerMon.Tomato.TON(pt := #Param.timerMon.Tomato.PT, et =>)
   END_RUNG
   RUNG wire#w1
      Contact( #Param.timerMon.Tomato.Q )
      S_Coil( #AlarmFlow_Blend.%X3 )
   END_RUNG
   // the same network as SCL:
   #Param.timerMon.Tomato.TON(IN := #alwaysON AND "T-05_Tomato".IN_Dose_Run AND NOT "T-05_Tomato".IN_Dose_Held AND "T-05_Tomato".IN_Dose_Pump_Cmd AND ("Totalizer_FT-05.01".value < #Param.min_Flow.Tomato),
                           PT := #Param.timerMon.Tomato.PT);
   IF #alwaysON AND #Param.timerMon.Tomato.Q THEN #AlarmFlow_Blend.%X3 := TRUE; END_IF;
END_REGION

REGION Network 7: Alarm Flow ChiliFresh 1
   RUNG wire#powerrail
      Contact( #alwaysON )
      wire#w1
      Contact( "T-06_ChiliFresh_1".IN_Dose_Run )
      I_Contact( "T-06_ChiliFresh_1".IN_Dose_Held )
      Contact( "T-06_ChiliFresh_1".IN_Dose_Pump_Cmd )
      { S7_Templates := "SrcType := Real" } LT_Contact(in1 := "Totalizer_FT-06.01".value, in2 := #Param.min_Flow.ChiliFresh1)
      { S7_Templates := "time_type := Time" } #Param.timerMon.ChiliFresh1.TON(pt := #Param.timerMon.ChiliFresh1.PT, et =>)
   END_RUNG
   RUNG wire#w1
      Contact( #Param.timerMon.ChiliFresh1.Q )
      S_Coil( #AlarmFlow_Blend.%X4 )
   END_RUNG
   // the same network as SCL:
   #Param.timerMon.ChiliFresh1.TON(IN := #alwaysON AND "T-06_ChiliFresh_1".IN_Dose_Run AND NOT "T-06_ChiliFresh_1".IN_Dose_Held AND "T-06_ChiliFresh_1".IN_Dose_Pump_Cmd AND ("Totalizer_FT-06.01".value < #Param.min_Flow.ChiliFresh1),
                           PT := #Param.timerMon.ChiliFresh1.PT);
   IF #alwaysON AND #Param.timerMon.ChiliFresh1.Q THEN #AlarmFlow_Blend.%X4 := TRUE; END_IF;
END_REGION

REGION Network 8: Alarm Flow ChiliFresh 2
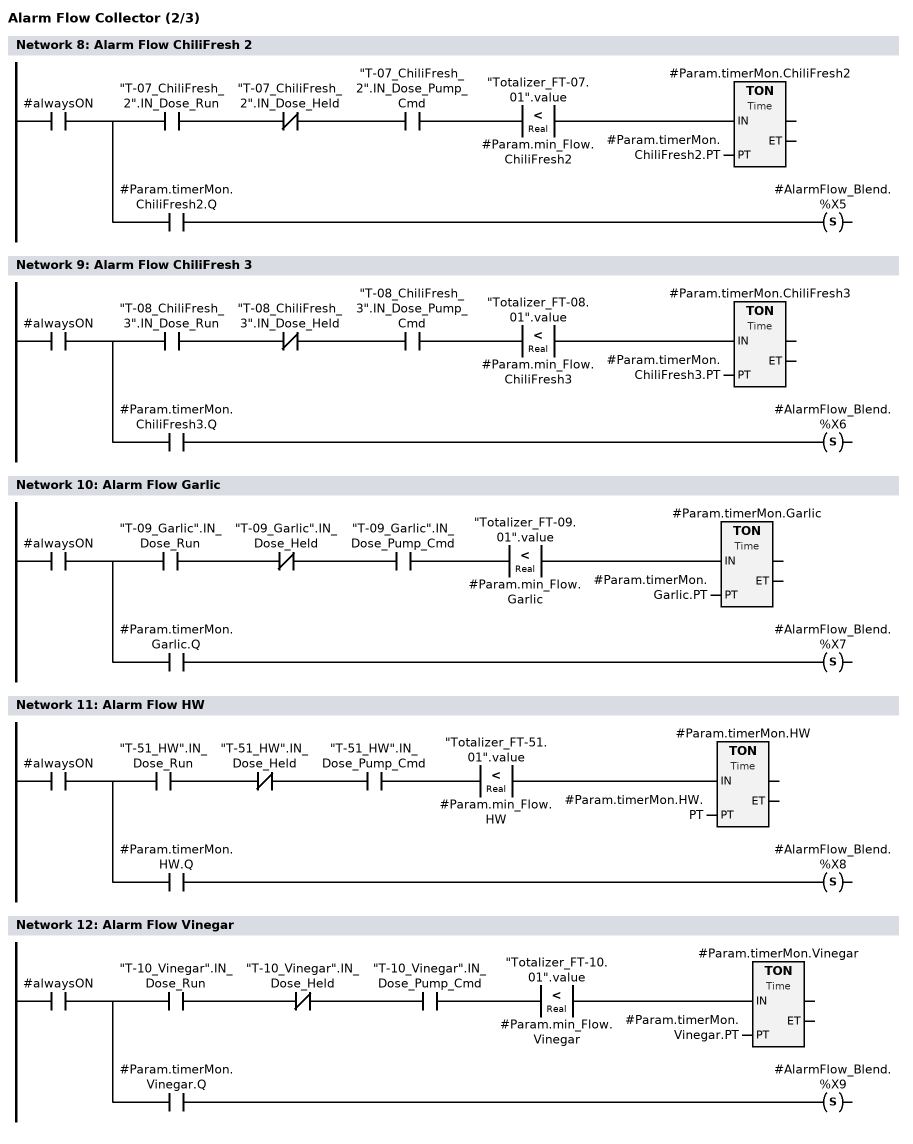
   RUNG wire#powerrail
      Contact( #alwaysON )
      wire#w1
      Contact( "T-07_ChiliFresh_2".IN_Dose_Run )
      I_Contact( "T-07_ChiliFresh_2".IN_Dose_Held )
      Contact( "T-07_ChiliFresh_2".IN_Dose_Pump_Cmd )
      { S7_Templates := "SrcType := Real" } LT_Contact(in1 := "Totalizer_FT-07.01".value, in2 := #Param.min_Flow.ChiliFresh2)
      { S7_Templates := "time_type := Time" } #Param.timerMon.ChiliFresh2.TON(pt := #Param.timerMon.ChiliFresh2.PT, et =>)
   END_RUNG
   RUNG wire#w1
      Contact( #Param.timerMon.ChiliFresh2.Q )
      S_Coil( #AlarmFlow_Blend.%X5 )
   END_RUNG
   // the same network as SCL:
   #Param.timerMon.ChiliFresh2.TON(IN := #alwaysON AND "T-07_ChiliFresh_2".IN_Dose_Run AND NOT "T-07_ChiliFresh_2".IN_Dose_Held AND "T-07_ChiliFresh_2".IN_Dose_Pump_Cmd AND ("Totalizer_FT-07.01".value < #Param.min_Flow.ChiliFresh2),
                           PT := #Param.timerMon.ChiliFresh2.PT);
   IF #alwaysON AND #Param.timerMon.ChiliFresh2.Q THEN #AlarmFlow_Blend.%X5 := TRUE; END_IF;
END_REGION

REGION Network 9: Alarm Flow ChiliFresh 3
   RUNG wire#powerrail
      Contact( #alwaysON )
      wire#w1
      Contact( "T-08_ChiliFresh_3".IN_Dose_Run )
      I_Contact( "T-08_ChiliFresh_3".IN_Dose_Held )
      Contact( "T-08_ChiliFresh_3".IN_Dose_Pump_Cmd )
      { S7_Templates := "SrcType := Real" } LT_Contact(in1 := "Totalizer_FT-08.01".value, in2 := #Param.min_Flow.ChiliFresh3)
      { S7_Templates := "time_type := Time" } #Param.timerMon.ChiliFresh3.TON(pt := #Param.timerMon.ChiliFresh3.PT, et =>)
   END_RUNG
   RUNG wire#w1
      Contact( #Param.timerMon.ChiliFresh3.Q )
      S_Coil( #AlarmFlow_Blend.%X6 )
   END_RUNG
   // the same network as SCL:
   #Param.timerMon.ChiliFresh3.TON(IN := #alwaysON AND "T-08_ChiliFresh_3".IN_Dose_Run AND NOT "T-08_ChiliFresh_3".IN_Dose_Held AND "T-08_ChiliFresh_3".IN_Dose_Pump_Cmd AND ("Totalizer_FT-08.01".value < #Param.min_Flow.ChiliFresh3),
                           PT := #Param.timerMon.ChiliFresh3.PT);
   IF #alwaysON AND #Param.timerMon.ChiliFresh3.Q THEN #AlarmFlow_Blend.%X6 := TRUE; END_IF;
END_REGION

REGION Network 10: Alarm Flow Garlic
   RUNG wire#powerrail
      Contact( #alwaysON )
      wire#w1
      Contact( "T-09_Garlic".IN_Dose_Run )
      I_Contact( "T-09_Garlic".IN_Dose_Held )
      Contact( "T-09_Garlic".IN_Dose_Pump_Cmd )
      { S7_Templates := "SrcType := Real" } LT_Contact(in1 := "Totalizer_FT-09.01".value, in2 := #Param.min_Flow.Garlic)
      { S7_Templates := "time_type := Time" } #Param.timerMon.Garlic.TON(pt := #Param.timerMon.Garlic.PT, et =>)
   END_RUNG
   RUNG wire#w1
      Contact( #Param.timerMon.Garlic.Q )
      S_Coil( #AlarmFlow_Blend.%X7 )
   END_RUNG
   // the same network as SCL:
   #Param.timerMon.Garlic.TON(IN := #alwaysON AND "T-09_Garlic".IN_Dose_Run AND NOT "T-09_Garlic".IN_Dose_Held AND "T-09_Garlic".IN_Dose_Pump_Cmd AND ("Totalizer_FT-09.01".value < #Param.min_Flow.Garlic),
                           PT := #Param.timerMon.Garlic.PT);
   IF #alwaysON AND #Param.timerMon.Garlic.Q THEN #AlarmFlow_Blend.%X7 := TRUE; END_IF;
END_REGION

REGION Network 11: Alarm Flow HW
   RUNG wire#powerrail
      Contact( #alwaysON )
      wire#w1
      Contact( "T-51_HW".IN_Dose_Run )
      I_Contact( "T-51_HW".IN_Dose_Held )
      Contact( "T-51_HW".IN_Dose_Pump_Cmd )
      { S7_Templates := "SrcType := Real" } LT_Contact(in1 := "Totalizer_FT-51.01".value, in2 := #Param.min_Flow.HW)
      { S7_Templates := "time_type := Time" } #Param.timerMon.HW.TON(pt := #Param.timerMon.HW.PT, et =>)
   END_RUNG
   RUNG wire#w1
      Contact( #Param.timerMon.HW.Q )
      S_Coil( #AlarmFlow_Blend.%X8 )
   END_RUNG
   // the same network as SCL:
   #Param.timerMon.HW.TON(IN := #alwaysON AND "T-51_HW".IN_Dose_Run AND NOT "T-51_HW".IN_Dose_Held AND "T-51_HW".IN_Dose_Pump_Cmd AND ("Totalizer_FT-51.01".value < #Param.min_Flow.HW),
                          PT := #Param.timerMon.HW.PT);
   IF #alwaysON AND #Param.timerMon.HW.Q THEN #AlarmFlow_Blend.%X8 := TRUE; END_IF;
END_REGION

REGION Network 12: Alarm Flow Vinegar
   RUNG wire#powerrail
      Contact( #alwaysON )
      wire#w1
      Contact( "T-10_Vinegar".IN_Dose_Run )
      I_Contact( "T-10_Vinegar".IN_Dose_Held )
      Contact( "T-10_Vinegar".IN_Dose_Pump_Cmd )
      { S7_Templates := "SrcType := Real" } LT_Contact(in1 := "Totalizer_FT-10.01".value, in2 := #Param.min_Flow.Vinegar)
      { S7_Templates := "time_type := Time" } #Param.timerMon.Vinegar.TON(pt := #Param.timerMon.Vinegar.PT, et =>)
   END_RUNG
   RUNG wire#w1
      Contact( #Param.timerMon.Vinegar.Q )
      S_Coil( #AlarmFlow_Blend.%X9 )
   END_RUNG
   // the same network as SCL:
   #Param.timerMon.Vinegar.TON(IN := #alwaysON AND "T-10_Vinegar".IN_Dose_Run AND NOT "T-10_Vinegar".IN_Dose_Held AND "T-10_Vinegar".IN_Dose_Pump_Cmd AND ("Totalizer_FT-10.01".value < #Param.min_Flow.Vinegar),
                           PT := #Param.timerMon.Vinegar.PT);
   IF #alwaysON AND #Param.timerMon.Vinegar.Q THEN #AlarmFlow_Blend.%X9 := TRUE; END_IF;
END_REGION

REGION Network 13: Alarm Flow Sugar
END_REGION

REGION Network 14: Alarm Flow Salt
END_REGION

REGION Network 15: Alarm Flow Prowater
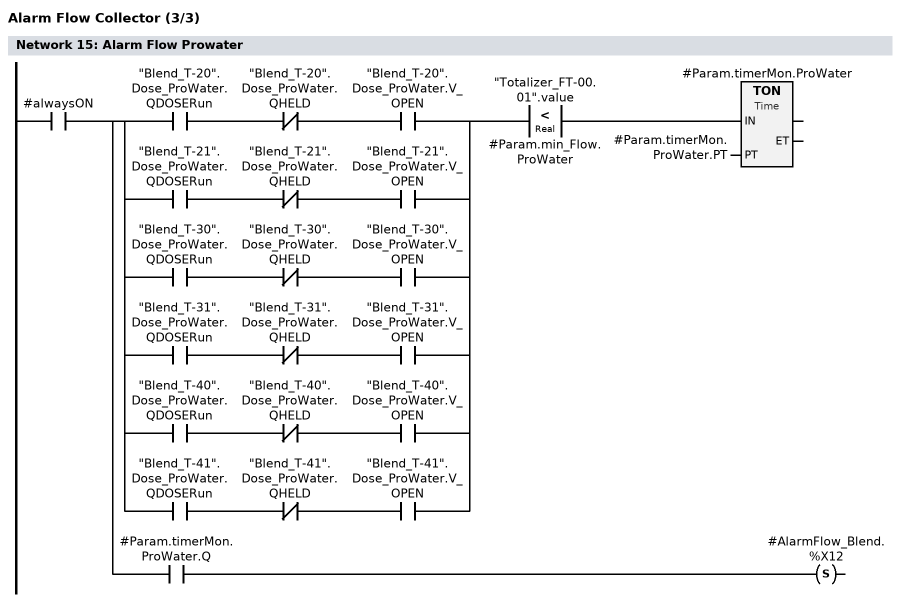
   RUNG wire#powerrail
      Contact( #alwaysON )
      wire#w1
      Contact( "Blend_T-20".Dose_ProWater.QDOSERun )
      I_Contact( "Blend_T-20".Dose_ProWater.QHELD )
      Contact( "Blend_T-20".Dose_ProWater.V_OPEN )
      wire#w2
      { S7_Templates := "SrcType := Real" } LT_Contact(in1 := "Totalizer_FT-00.01".value, in2 := #Param.min_Flow.ProWater)
      { S7_Templates := "time_type := Time" } #Param.timerMon.ProWater.TON(pt := #Param.timerMon.ProWater.PT, et =>)
   END_RUNG
   RUNG wire#w1
      Contact( "Blend_T-21".Dose_ProWater.QDOSERun )
      I_Contact( "Blend_T-21".Dose_ProWater.QHELD )
      Contact( "Blend_T-21".Dose_ProWater.V_OPEN )
   END_RUNG wire#w2
   RUNG wire#w1
      Contact( "Blend_T-30".Dose_ProWater.QDOSERun )
      I_Contact( "Blend_T-30".Dose_ProWater.QHELD )
      Contact( "Blend_T-30".Dose_ProWater.V_OPEN )
   END_RUNG wire#w2
   RUNG wire#w1
      Contact( "Blend_T-31".Dose_ProWater.QDOSERun )
      I_Contact( "Blend_T-31".Dose_ProWater.QHELD )
      Contact( "Blend_T-31".Dose_ProWater.V_OPEN )
   END_RUNG wire#w2
   RUNG wire#w1
      Contact( "Blend_T-40".Dose_ProWater.QDOSERun )
      I_Contact( "Blend_T-40".Dose_ProWater.QHELD )
      Contact( "Blend_T-40".Dose_ProWater.V_OPEN )
   END_RUNG wire#w2
   RUNG wire#w1
      Contact( "Blend_T-41".Dose_ProWater.QDOSERun )
      I_Contact( "Blend_T-41".Dose_ProWater.QHELD )
      Contact( "Blend_T-41".Dose_ProWater.V_OPEN )
   END_RUNG wire#w2
   RUNG wire#w1
      Contact( #Param.timerMon.ProWater.Q )
      S_Coil( #AlarmFlow_Blend.%X12 )
   END_RUNG
   // the same network as SCL:
   #Param.timerMon.ProWater.TON(IN := #alwaysON AND (("Blend_T-20".Dose_ProWater.QDOSERun AND NOT "Blend_T-20".Dose_ProWater.QHELD AND "Blend_T-20".Dose_ProWater.V_OPEN) OR ("Blend_T-21".Dose_ProWater.QDOSERun AND NOT "Blend_T-21".Dose_ProWater.QHELD AND "Blend_T-21".Dose_ProWater.V_OPEN) OR ("Blend_T-30".Dose_ProWater.QDOSERun AND NOT "Blend_T-30".Dose_ProWater.QHELD AND "Blend_T-30".Dose_ProWater.V_OPEN) OR ("Blend_T-31".Dose_ProWater.QDOSERun AND NOT "Blend_T-31".Dose_ProWater.QHELD AND "Blend_T-31".Dose_ProWater.V_OPEN) OR ("Blend_T-40".Dose_ProWater.QDOSERun AND NOT "Blend_T-40".Dose_ProWater.QHELD AND "Blend_T-40".Dose_ProWater.V_OPEN) OR ("Blend_T-41".Dose_ProWater.QDOSERun AND NOT "Blend_T-41".Dose_ProWater.QHELD AND "Blend_T-41".Dose_ProWater.V_OPEN)) AND ("Totalizer_FT-00.01".value < #Param.min_Flow.ProWater),
                           PT := #Param.timerMon.ProWater.PT);
   IF #alwaysON AND #Param.timerMon.ProWater.Q THEN #AlarmFlow_Blend.%X12 := TRUE; END_IF;
END_REGION
END_FUNCTION_BLOCK

FUNCTION_BLOCK "Blend_Tank"   // FB210, LAD
{ S7_Optimized_Access := 'TRUE' }
VERSION : 0.1
// stored: AutoNumber false, IsIECCheckEnabled false, IsRetainMemResEnabled false, MemoryReserve 100, SetENOAutomatically false, UDAEnableTagReadback false
   VAR_INPUT
      IN_FBAV_Header1 : Bool;
      IN_FBAV_Header2 : Bool;
      IN_FBAV_Vinegar : Bool;
      IN_FBAV_Sugar : Bool;
      IN_FBAV_Salt : Bool;
      IN_FBAV_ProWater : Bool;
      IN_FBAV_Homomixer : Bool;
      IN_FBAV_Transfer1 : Bool;
      IN_FBAV_Transfer2 : Bool;
      IN_FBAV_Transfer3 : Bool;
      IN_FBAV_Outlet : Bool;
      IN_FBAV_CIP : Bool;
      IN_FBP_Transfer1 : Bool;
      IN_FBP_Transfer1_Sp : Real;
      IN_FBP_Transfer2 : Bool;
      IN_FBP_Transfer2_Sp : Real;
      IN_FBP_Transfer3 : Bool;
      IN_FBP_Transfer3_Sp : Real;
      IN_FBP_CIP : Bool;
      IN_FBP_CIP_Sp : Real;
      IN_LT01 : Real;
      "BFT-1 Prod Req" : Bool;
      "BFT-1 Prod Line" : Bool;
      "BFT-1 CIP Enable" : Bool;
      "BFT-1 CIPLine" : Bool;
      "BFT-2 Prod Req" : Bool;
      "BFT-2 Prod Line" : Bool;
      "BFT-2 CIP Enable" : Bool;
      "BFT-2 CIPLine" : Bool;
      "BFT-3 Prod Req" : Bool;
      "BFT-3 Prod Line" : Bool;
      "BFT-3 CIP Enable" : Bool;
      "BFT-3 CIPLine" : Bool;
      "Transfer 1 Busy" : Bool;
      "Transfer 2 Busy" : Bool;
      "Transfer 3 Busy" : Bool;
      "Header 1 Available" : Bool;   // Header 1 line free
      "Header 2 Available" : Bool;   // Header 2 line free
      "Vinegar Available" : Bool;   // Vinegar line free
      "Sugar Available" : Bool;   // Sugar line free
      "Salt Available" : Bool;   // Salt line free
      "ProWater Available" : Bool;   // ProWater line free
      "Homomixer Available" : Bool;   // Homomixer line free
      IN_LDT : Date_And_Time;
      "CIP Pulse" : Bool;
      "CIP Supply ON" : Bool;
      "CIP Req OK" : Bool;
      "CIP Complete" : Bool;
      "CIP Busy" : Bool;
   END_VAR
   VAR_OUTPUT
      Out_AV_Header1 : Bool;
      Out_AV_Header2 : Bool;
      Out_AV_Vinegar : Bool;
      Out_AV_Sugar : Bool;
      Out_AV_Salt : Bool;
      Out_AV_ProWater : Bool;
      Out_AV_Homomixer : Bool;
      Out_AV_Transfer1 : Bool;
      Out_AV_Transfer2 : Bool;
      Out_AV_Transfer3 : Bool;
      Out_AV_Outlet : Bool;
      Out_AV_CIP : Bool;
      Out_P_Transfer1 : Bool;
      Out_P_Transfer1_Sp : Real;
      Out_P_Transfer2 : Bool;
      Out_P_Transfer2_Sp : Real;
      Out_P_Transfer3 : Bool;
      Out_P_Transfer3_Sp : Real;
      Out_P_CIP : Bool;
      Out_P_CIP_Sp : Real;
      Out_Agi : Bool;
      Out_Agi_Sp : Real;
      "Header 1 Req" : Bool;
      "Header 2 Req" : Bool;
      "Vinegar Req" : Bool;
      "Sugar Req" : Bool;
      "Salt Req" : Bool;
      "ProWater Req" : Bool;
      "Homomixer Req" : Bool;
      Out_CIP_Req : Bool;
      Out_CIP_Line_Open : Bool;
   END_VAR
   VAR
      Cmd : Struct
         "Ready For Transfer" : Bool;
         "CIP Tank 1" : Bool;
         "CIP Tank 2" : Bool;
         "CIP Line" : Bool;
         "Dose Head 1" : Bool;
         "Dose Head 2" : Bool;
         Agitator_Mode : Bool;   // 0: Speed Fix, 1: Speed by level
      END_STRUCT;
   END_VAR
   VAR RETAIN
      Param : Struct
         SP_Level_LL : Real := 10.0;
         SP_Level_ML : Real := 80.0;
         SP_Level_HL : Real := 100.0;
         L_Hi_Lim : Real := 100.0;
         L_Lo_Lim : Real := 0.0;
         L_Hys : Real := 2.0;
         LB_ON : Real := 20.0;
         LB_OFF : Real := 17.0;
         LB1_ON : Real := 15.0;
         LB1_OFF : Real := 10.0;
         LB2_ON : Real := 35.0;
         LB2_OFF : Real := 30.0;
         LB3_ON : Real := 65.0;
         LB3_OFF : Real := 60.0;
         SP_P1_Speed : Real := 80.0;
         SP_P2_Speed : Real := 80.0;
         SP_P3_Speed : Real := 80.0;
         SP_LB_Speed : Real := 50.0;
         SP_LB1_Speed : Real := 25.0;
         SP_LB2_Speed : Real := 50.0;
         SP_LB3_Speed : Real := 80.0;
         CIP_Tank_P_Ret_Speed : Real := 60.0;
         CIP_Ret_ON_SP : Real := 10.0;
         CIP_Ret_OFF_SP : Real := 0.0;
         Flushing_HW_Timer : Time := T#60s;
      END_STRUCT;
   END_VAR
   VAR
      State : Struct
         "Tank LL" : Bool;
         "Tank ML" : Bool;
         "Tank HL" : Bool;
         LB_ON : Bool;
         LB1_ON : Bool;
         LB2_ON : Bool;
         LB3_ON : Bool;
         "CIP Tank" : Bool;
         "CIP Tank Ena" : Bool;
         "CIP Tank Ret 1 Ena" : Bool;
         "CIP Tank Ret 2 Ena" : Bool;
         "CIP Line" : Bool;
         "CIP Line Ena" : Bool;
         "CIP Return On" : Bool;
         "Dose On Prog" : Bool;
         "Dose EN" : Bool;
         "Ready For Transfer" : Bool;
         "Ready For Transfer Ena" : Bool;
         "BFT-1 EN" : Bool;
         "BFT-2 EN" : Bool;
         "BFT-3 EN" : Bool;
         "RM Dose" : Bool;
         "Transfer 1 On Progress" : Bool;
         "Transfer 2 On Progress" : Bool;
         "Transfer 3 On Progress" : Bool;
         "DoseHead1 ON" : Bool;
         "DoseHead2 ON" : Bool;
      END_STRUCT;
      Dose : Struct
         Dose_Start : DWord;
         Dose_Pause : DWord;
         Dose_Stop : DWord;
         Dose_State : DWord;
         Dose_Tank_Available : Word;
         Dose_Prod_Ready : Word;
         Dose_Header_Req : DWord;
         Dose_EN : Word;
      END_STRUCT;
      "Dose_Level_%" : Struct
         "ChiliAwetan1%" : Real;
         "ChiliAwetan2%" : Real;
         "ChiliAwetan3%" : Real;
         "Tomato%" : Real;
         "ChiliFresh1%" : Real;
         "ChiliFresh2%" : Real;
         "ChiliFresh3%" : Real;
         "Garlic%" : Real;
         "HW%" : Real;
         "Vinegar%" : Real;
         "Sugar%" : Real;
         "Salt%" : Real;
         "ProWater%" : Real;
         "Homomixer%" : Real;
      END_STRUCT;
      Dose_Level_Lit : Struct
         ChiliAwetan1Lit : Real;
         ChiliAwetan2Lit : Real;
         ChiliAwetan3Lit : Real;
         TomatoLit : Real;
         ChiliFresh1Lit : Real;
         ChiliFresh2Lit : Real;
         ChiliFresh3Lit : Real;
         GarlicLit : Real;
         HWLit : Real;
         VinegarLit : Real;
         SugarLit : Real;
         SaltLit : Real;
         ProWaterLit : Real;
         HomomixerLit : Real;
      END_STRUCT;
      SP_Dose_Level : Struct
         ChiliAwetan1Lit : Real;
         ChiliAwetan2Lit : Real;
         ChiliAwetan3Lit : Real;
         TomatoLit : Real;
         ChiliFresh1Lit : Real;
         ChiliFresh2Lit : Real;
         ChiliFresh3Lit : Real;
         GarlicLit : Real;
         HWLit : Real;
         VinegarLit : Real;
         SugarLit : Real;
         SaltLit : Real;
         ProWaterLit : Real;
         HomomixerLit : Real;
      END_STRUCT;
      r : Struct
         PosE1 : Bool;
         PosE2 : Bool;
         PosE3 : Bool;
         PosE4 : Bool;
         PosE5 : Bool;
         PosE6 : Bool;
         PosE7 : Bool;
         PosE8 : Bool;
         PosE9 : Bool;
         PosE10 : Bool;
         PosE11 : Bool;
         PosE12 : Bool;
         PosE13 : Bool;
         PosE14 : Bool;
         PosE15 : Bool;
         PosE16 : Bool;
         PosE17 : Bool;
         PosE18 : Bool;
         PosE19 : Bool;
         PosE20 : Bool;
         PosE21 : Bool;
         PosE22 : Bool;
         PosE23 : Bool;
         PosE24 : Bool;
         PosE25 : Bool;
         PosE26 : Bool;
         PosE27 : Bool;
         PosE28 : Bool;
         PosE29 : Bool;
         PosE30 : Bool;
         PosE31 : Bool;
         PosE32 : Bool;
      END_STRUCT;
      Actuator : Struct
         P_Transfer1 : Bool;
         P_Transfer2 : Bool;
         P_Transfer3 : Bool;
         AV_Transfer1 : Bool;
         AV_Transfer2 : Bool;
         AV_Transfer3 : Bool;
         AV_Outlet : Bool;
         AV_CIP_Tank : Bool;
      END_STRUCT;
      SP_ChiliAwetan1 : "RawDose";
      SP_ChiliAwetan2 : "RawDose";
      SP_ChiliAwetan3 : "RawDose";
      SP_Tomato : "RawDose";
      SP_ChiliFresh1 : "RawDose";
      SP_ChiliFresh2 : "RawDose";
      SP_ChiliFresh3 : "RawDose";
      SP_Garlic : "RawDose";
      SP_HW : "Raw_Pulse";
      SP_Vinegar : "RawDose";
      SP_Sugar : "RawDose";
      SP_Salt : "RawDose";
      SP_ProWater : "Raw_Pulse";
      SP_Homomixer : "RawDose";
      Dose_ChiliAwetan1 { S7_SetPoint := 'True'} : "DOSE";
      Dose_ChiliAwetan2 { S7_SetPoint := 'True'} : "DOSE";
      Dose_ChiliAwetan3 { S7_SetPoint := 'True'} : "DOSE";
      Dose_Tomato { S7_SetPoint := 'True'} : "DOSE";
      Dose_ChiliFresh1 { S7_SetPoint := 'True'} : "DOSE";
      Dose_ChiliFresh2 { S7_SetPoint := 'True'} : "DOSE";
      Dose_ChiliFresh3 { S7_SetPoint := 'True'} : "DOSE";
      Dose_Garlic { S7_SetPoint := 'True'} : "DOSE";
      Dose_HW { S7_SetPoint := 'True'} : "DOSE";
      Dose_Vinegar { S7_SetPoint := 'True'} : "DOSE";
      Dose_Sugar { S7_SetPoint := 'True'} : "DOSE";
      Dose_Salt { S7_SetPoint := 'True'} : "DOSE";
      Dose_ProWater { S7_SetPoint := 'True'} : "DOSE";
      Dose_Homomixer { S7_SetPoint := 'True'} : "DOSE";
      AlwaysON { S7_SetPoint := 'True'} : Bool;
      L_Hys_Abs { S7_SetPoint := 'True'} : Real;
      Hys_Level_HL : Real;
      Hys_Level_ML : Real;
      Hys_Level_LL : Real;
      TimerOff_Valve_Out : TON_TIME;
      TimerOff_Valve_P_1 { S7_SetPoint := 'True'} : TON_TIME;
      TimerOff_Valve_P_2 { S7_SetPoint := 'True'} : TON_TIME;
      TimerOff_Valve_P_3 { S7_SetPoint := 'True'} : TON_TIME;
      TimerOff_Valve_P_CIP { S7_SetPoint := 'True'} : TON_TIME;
   END_VAR
   VAR RETAIN
      Last_Dose_Qty : Struct
         ChiliAwetan1 : Real;
         ChiliAwetan2 : Real;
         ChiliAwetan3 : Real;
         Tomato : Real;
         ChiliFresh1 : Real;
         ChiliFresh2 : Real;
         ChiliFresh3 : Real;
         Garlic : Real;
         HW : Real;
         Vinegar : Real;
         Sugar : Real;
         Salt : Real;
         ProWater : Real;
         Homomixer : Real;
      END_STRUCT;
   END_VAR
   VAR
      "HW Flushing" : Struct
         Status : Struct
            "Flush to Blend" : Bool;
            "Flush to Drain" : Bool;
            Drain : Bool;
            Done : Bool;
         END_STRUCT;
         Qty : Struct
            "Flush to Blend Qty" : Real;
            "Flush to Drain Qty" : Real;
            "Flush to Blend Act" : Real;
            "Flush to Drain Act" : Real;
         END_STRUCT;
         TimeDrain_SP : DInt;
         Cmd_Start_Drain : Bool;
         Cmd_Stop_Drain : Bool;
         DrainTime : TONR_TIME;
      END_STRUCT;
      PumpTF1_OnDelay : TON_TIME;
      PumpTF2_OnDelay { S7_SetPoint := 'True'} : TON_TIME;
      PumpTF3_OnDelay { S7_SetPoint := 'True'} : TON_TIME;
   END_VAR
   VAR RETAIN
      TimerON : Struct
         TimerON_1 : TON_TIME;
         TimerON_2 { S7_SetPoint := 'True'} : TON_TIME;
         TimerON_3 { S7_SetPoint := 'True'} : TON_TIME;
         TimerON_4 { S7_SetPoint := 'True'} : TON_TIME;
         TimerON_5 { S7_SetPoint := 'True'} : TON_TIME;
         TimerON_6 { S7_SetPoint := 'True'} : TON_TIME;
         TimerON_7 { S7_SetPoint := 'True'} : TON_TIME;
         TimerON_8 { S7_SetPoint := 'True'} : TON_TIME;
      END_STRUCT;
      TimerOFF : Struct
         TimerOFF_1 : TOF_TIME;
         TimerOFF_2 { S7_SetPoint := 'True'} : TOF_TIME;
         TimerOFF_3 { S7_SetPoint := 'True'} : TOF_TIME;
         TimerOFF_4 { S7_SetPoint := 'True'} : TOF_TIME;
         TimerOFF_5 { S7_SetPoint := 'True'} : TOF_TIME;
         TimerOFF_6 { S7_SetPoint := 'True'} : TOF_TIME;
         TimerOFF_7 { S7_SetPoint := 'True'} : TOF_TIME;
         TimerOFF_8 { S7_SetPoint := 'True'} : TOF_TIME;
      END_STRUCT;
   END_VAR
   // SP_ProWater.Para."SP_Qty_Fine%" := 10.0;
   // SP_Homomixer.Dose_SP := 10.0;
   // TimerON.TimerON_1.PT := T#8s;
   // TimerON.TimerON_2.PT := T#8s;
   // TimerON.TimerON_3.PT := T#10s;
   // TimerON.TimerON_4.PT := T#10s;
   // TimerON.TimerON_5.PT := T#10s;
   // TimerON.TimerON_6.PT := T#10s;
   // TimerON.TimerON_7.PT := T#10s;
   // TimerON.TimerON_8.PT := T#10s;
   // TimerOFF.TimerOFF_1.PT := T#10s;
   // TimerOFF.TimerOFF_2.PT := T#10s;
   // TimerOFF.TimerOFF_3.PT := T#10s;
   // TimerOFF.TimerOFF_4.PT := T#10s;
   // TimerOFF.TimerOFF_5.PT := T#10s;
   // TimerOFF.TimerOFF_6.PT := T#10s;
   // TimerOFF.TimerOFF_7.PT := T#10s;
   // TimerOFF.TimerOFF_8.PT := T#10s;
   VAR_TEMP   // added for the SCL form of the ladder/FBD networks
      _w1 : Bool;
      _w2 : Bool;
      _w3 : Bool;
      _w4 : Bool;
      _w5 : Bool;
      _w6 : Bool;
   END_VAR
BEGIN

REGION Network 2: Always ON
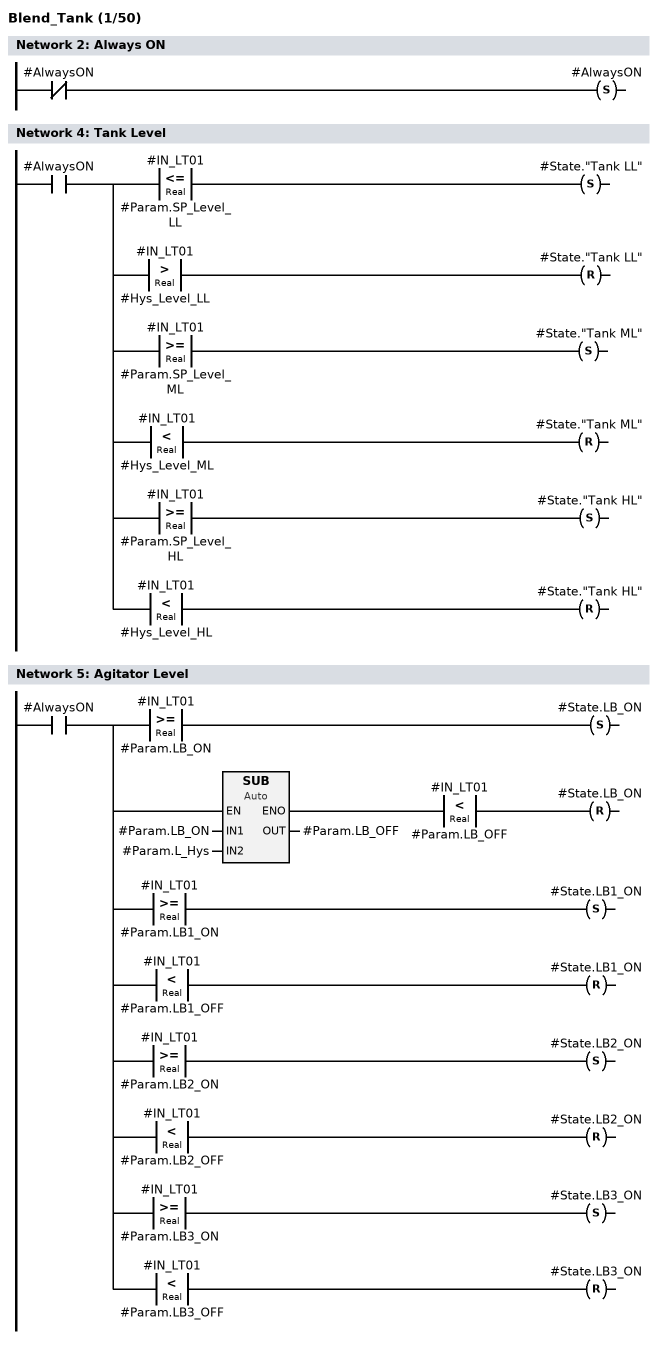
   RUNG wire#powerrail
      I_Contact( #AlwaysON )
      S_Coil( #AlwaysON )
   END_RUNG
   // the same network as SCL:
   IF NOT #AlwaysON THEN #AlwaysON := TRUE; END_IF;
END_REGION

NETWORK
TITLE = Hys Calculation
//Level Hys Absolute
      L     #Param.L_Hi_Lim;
      L     #Param.L_Lo_Lim;
      -R;
      L     100.0;
      /R;
      L     #Param.L_Hys;
      *R;
      T     #L_Hys_Abs;
//Tank High Level
      L     #Param.SP_Level_HL;
      L     #L_Hys_Abs;
      -R;
      T     #Hys_Level_HL;
//Tank Mid Level
      L     #Param.SP_Level_ML;
      L     #L_Hys_Abs;
      -R;
      T     #Hys_Level_ML;
//Tank Low Level
      L     #Param.SP_Level_LL;
      L     #L_Hys_Abs;
      +R;
      T     #Hys_Level_LL;


REGION Network 4: Tank Level
   RUNG wire#powerrail
      Contact( #AlwaysON )
      wire#w1
      { S7_Templates := "SrcType := Real" } LE_Contact(in1 := #IN_LT01, in2 := #Param.SP_Level_LL)
      S_Coil( #State."Tank LL" )
   END_RUNG
   RUNG wire#w1
      { S7_Templates := "SrcType := Real" } GT_Contact(in1 := #IN_LT01, in2 := #Hys_Level_LL)
      R_Coil( #State."Tank LL" )
   END_RUNG
   RUNG wire#w1
      { S7_Templates := "SrcType := Real" } GE_Contact(in1 := #IN_LT01, in2 := #Param.SP_Level_ML)
      S_Coil( #State."Tank ML" )
   END_RUNG
   RUNG wire#w1
      { S7_Templates := "SrcType := Real" } LT_Contact(in1 := #IN_LT01, in2 := #Hys_Level_ML)
      R_Coil( #State."Tank ML" )
   END_RUNG
   RUNG wire#w1
      { S7_Templates := "SrcType := Real" } GE_Contact(in1 := #IN_LT01, in2 := #Param.SP_Level_HL)
      S_Coil( #State."Tank HL" )
   END_RUNG
   RUNG wire#w1
      { S7_Templates := "SrcType := Real" } LT_Contact(in1 := #IN_LT01, in2 := #Hys_Level_HL)
      R_Coil( #State."Tank HL" )
   END_RUNG
   // the same network as SCL:
   IF #AlwaysON AND (#IN_LT01 <= #Param.SP_Level_LL) THEN #State."Tank LL" := TRUE; END_IF;
   IF #AlwaysON AND (#IN_LT01 > #Hys_Level_LL) THEN #State."Tank LL" := FALSE; END_IF;
   IF #AlwaysON AND (#IN_LT01 >= #Param.SP_Level_ML) THEN #State."Tank ML" := TRUE; END_IF;
   IF #AlwaysON AND (#IN_LT01 < #Hys_Level_ML) THEN #State."Tank ML" := FALSE; END_IF;
   IF #AlwaysON AND (#IN_LT01 >= #Param.SP_Level_HL) THEN #State."Tank HL" := TRUE; END_IF;
   IF #AlwaysON AND (#IN_LT01 < #Hys_Level_HL) THEN #State."Tank HL" := FALSE; END_IF;
END_REGION

REGION Network 5: Agitator Level
   RUNG wire#powerrail
      Contact( #AlwaysON )
      wire#w1
      { S7_Templates := "SrcType := Real" } GE_Contact(in1 := #IN_LT01, in2 := #Param.LB_ON)
      S_Coil( #State.LB_ON )
   END_RUNG
   RUNG wire#w1
      Sub(in1 := #Param.LB_ON, in2 := #Param.L_Hys, out => #Param.LB_OFF)
      { S7_Templates := "SrcType := Real" } LT_Contact(in1 := #IN_LT01, in2 := #Param.LB_OFF)
      R_Coil( #State.LB_ON )
   END_RUNG
   RUNG wire#w1
      { S7_Templates := "SrcType := Real" } GE_Contact(in1 := #IN_LT01, in2 := #Param.LB1_ON)
      S_Coil( #State.LB1_ON )
   END_RUNG
   RUNG wire#w1
      { S7_Templates := "SrcType := Real" } LT_Contact(in1 := #IN_LT01, in2 := #Param.LB1_OFF)
      R_Coil( #State.LB1_ON )
   END_RUNG
   RUNG wire#w1
      { S7_Templates := "SrcType := Real" } GE_Contact(in1 := #IN_LT01, in2 := #Param.LB2_ON)
      S_Coil( #State.LB2_ON )
   END_RUNG
   RUNG wire#w1
      { S7_Templates := "SrcType := Real" } LT_Contact(in1 := #IN_LT01, in2 := #Param.LB2_OFF)
      R_Coil( #State.LB2_ON )
   END_RUNG
   RUNG wire#w1
      { S7_Templates := "SrcType := Real" } GE_Contact(in1 := #IN_LT01, in2 := #Param.LB3_ON)
      S_Coil( #State.LB3_ON )
   END_RUNG
   RUNG wire#w1
      { S7_Templates := "SrcType := Real" } LT_Contact(in1 := #IN_LT01, in2 := #Param.LB3_OFF)
      R_Coil( #State.LB3_ON )
   END_RUNG
   // the same network as SCL:
   IF #AlwaysON AND (#IN_LT01 >= #Param.LB_ON) THEN #State.LB_ON := TRUE; END_IF;
   IF #AlwaysON THEN #Param.LB_OFF := #Param.LB_ON - #Param.L_Hys; END_IF;
   IF #AlwaysON AND (#IN_LT01 < #Param.LB_OFF) THEN #State.LB_ON := FALSE; END_IF;
   IF #AlwaysON AND (#IN_LT01 >= #Param.LB1_ON) THEN #State.LB1_ON := TRUE; END_IF;
   IF #AlwaysON AND (#IN_LT01 < #Param.LB1_OFF) THEN #State.LB1_ON := FALSE; END_IF;
   IF #AlwaysON AND (#IN_LT01 >= #Param.LB2_ON) THEN #State.LB2_ON := TRUE; END_IF;
   IF #AlwaysON AND (#IN_LT01 < #Param.LB2_OFF) THEN #State.LB2_ON := FALSE; END_IF;
   IF #AlwaysON AND (#IN_LT01 >= #Param.LB3_ON) THEN #State.LB3_ON := TRUE; END_IF;
   IF #AlwaysON AND (#IN_LT01 < #Param.LB3_OFF) THEN #State.LB3_ON := FALSE; END_IF;
END_REGION

REGION Network 6: Agitator ON-OFF
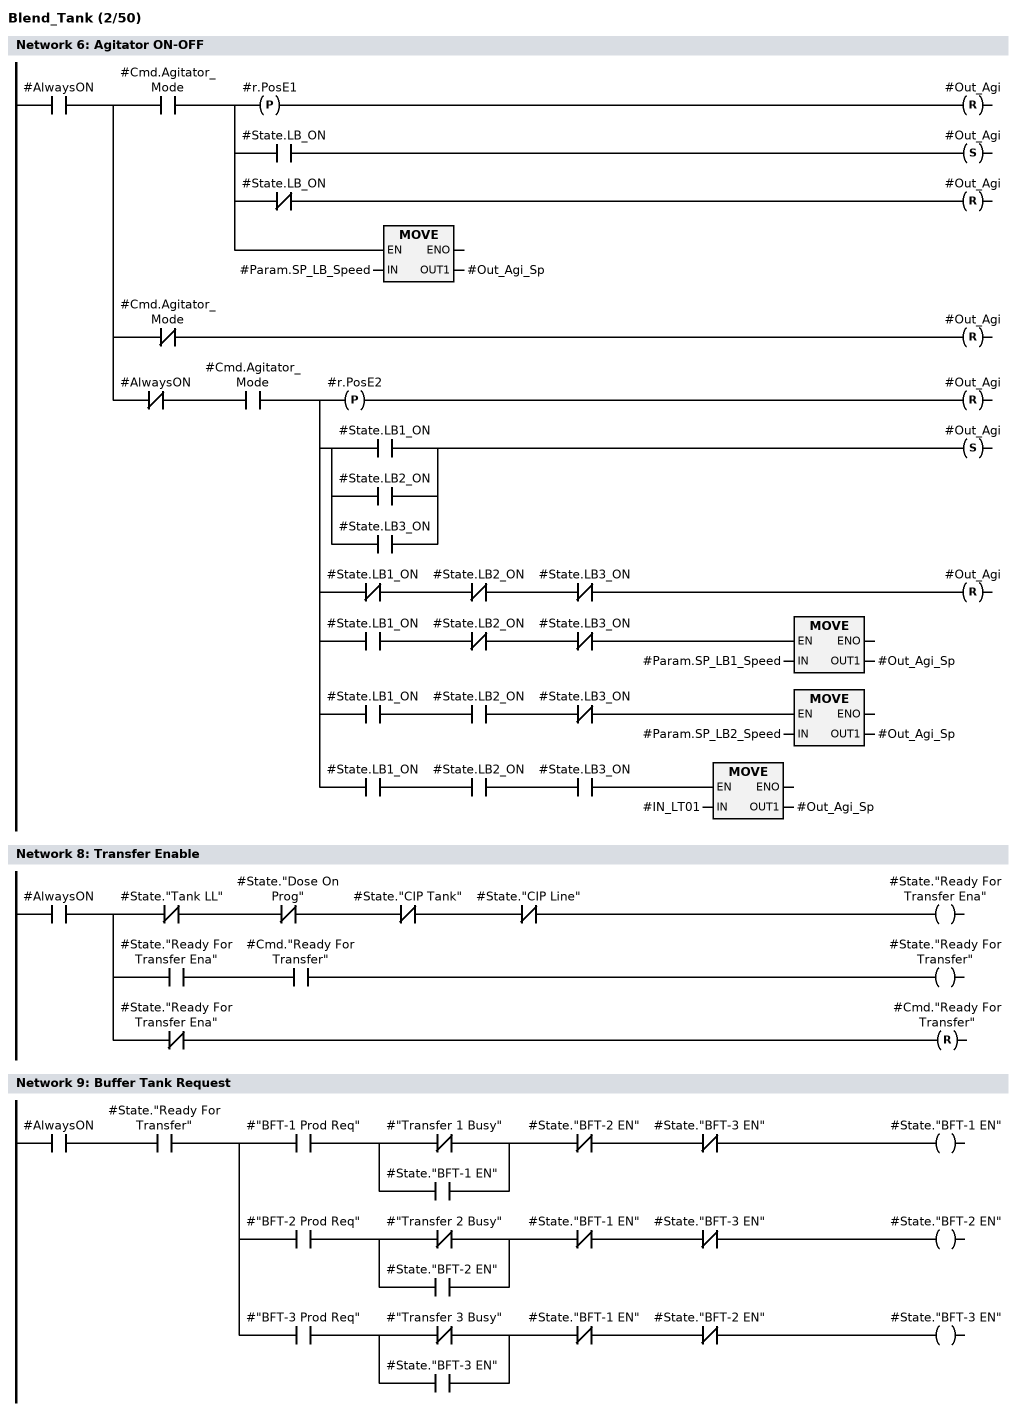
   RUNG wire#powerrail
      Contact( #AlwaysON )
      wire#w1
      Contact( #Cmd.Agitator_Mode )
      wire#w2
      P_Trig( #r.PosE1 )
      R_Coil( #Out_Agi )
   END_RUNG
   RUNG wire#w2
      Contact( #State.LB_ON )
      S_Coil( #Out_Agi )
   END_RUNG
   RUNG wire#w2
      I_Contact( #State.LB_ON )
      R_Coil( #Out_Agi )
   END_RUNG
   RUNG wire#w2
      Move(in := #Param.SP_LB_Speed, out1 => #Out_Agi_Sp)
   END_RUNG
   RUNG wire#w1
      I_Contact( #Cmd.Agitator_Mode )
      R_Coil( #Out_Agi )
   END_RUNG
   RUNG wire#w1
      I_Contact( #AlwaysON )
      Contact( #Cmd.Agitator_Mode )
      wire#w3
      P_Trig( #r.PosE2 )
      R_Coil( #Out_Agi )
   END_RUNG
   RUNG wire#w3
      Contact( #State.LB1_ON )
      wire#w4
      S_Coil( #Out_Agi )
   END_RUNG
   RUNG wire#w3
      Contact( #State.LB2_ON )
   END_RUNG wire#w4
   RUNG wire#w3
      Contact( #State.LB3_ON )
   END_RUNG wire#w4
   RUNG wire#w3
      I_Contact( #State.LB1_ON )
      I_Contact( #State.LB2_ON )
      I_Contact( #State.LB3_ON )
      R_Coil( #Out_Agi )
   END_RUNG
   RUNG wire#w3
      Contact( #State.LB1_ON )
      I_Contact( #State.LB2_ON )
      I_Contact( #State.LB3_ON )
      Move(in := #Param.SP_LB1_Speed, out1 => #Out_Agi_Sp)
   END_RUNG
   RUNG wire#w3
      Contact( #State.LB1_ON )
      Contact( #State.LB2_ON )
      I_Contact( #State.LB3_ON )
      Move(in := #Param.SP_LB2_Speed, out1 => #Out_Agi_Sp)
   END_RUNG
   RUNG wire#w3
      Contact( #State.LB1_ON )
      Contact( #State.LB2_ON )
      Contact( #State.LB3_ON )
      Move(in := #IN_LT01, out1 => #Out_Agi_Sp)
   END_RUNG
   // the same network as SCL:
   #_w1 := #AlwaysON AND #Cmd.Agitator_Mode;
   #_w2 := #_w1 AND NOT #r.PosE1;   // rising edge
   #r.PosE1 := #_w1;
   IF #_w2 THEN #Out_Agi := FALSE; END_IF;
   IF #_w1 AND #State.LB_ON THEN #Out_Agi := TRUE; END_IF;
   IF #_w1 AND NOT #State.LB_ON THEN #Out_Agi := FALSE; END_IF;
   IF #_w1 THEN #Out_Agi_Sp := #Param.SP_LB_Speed; END_IF;
   IF #AlwaysON AND NOT #Cmd.Agitator_Mode THEN #Out_Agi := FALSE; END_IF;
   #_w3 := #AlwaysON AND NOT #AlwaysON AND #Cmd.Agitator_Mode;
   #_w4 := #_w3 AND NOT #r.PosE2;   // rising edge
   #r.PosE2 := #_w3;
   IF #_w4 THEN #Out_Agi := FALSE; END_IF;
   IF #_w3 AND (#State.LB1_ON OR #State.LB2_ON OR #State.LB3_ON) THEN #Out_Agi := TRUE; END_IF;
   IF #_w3 AND NOT #State.LB1_ON AND NOT #State.LB2_ON AND NOT #State.LB3_ON THEN #Out_Agi := FALSE; END_IF;
   IF #_w3 AND #State.LB1_ON AND NOT #State.LB2_ON AND NOT #State.LB3_ON THEN
       #Out_Agi_Sp := #Param.SP_LB1_Speed;
   END_IF;
   IF #_w3 AND #State.LB1_ON AND #State.LB2_ON AND NOT #State.LB3_ON THEN
       #Out_Agi_Sp := #Param.SP_LB2_Speed;
   END_IF;
   IF #_w3 AND #State.LB1_ON AND #State.LB2_ON AND #State.LB3_ON THEN #Out_Agi_Sp := #IN_LT01; END_IF;
END_REGION

REGION Network 8: Transfer Enable
   RUNG wire#powerrail
      Contact( #AlwaysON )
      wire#w1
      I_Contact( #State."Tank LL" )
      I_Contact( #State."Dose On Prog" )
      I_Contact( #State."CIP Tank" )
      I_Contact( #State."CIP Line" )
      Coil( #State."Ready For Transfer Ena" )
   END_RUNG
   RUNG wire#w1
      Contact( #State."Ready For Transfer Ena" )
      Contact( #Cmd."Ready For Transfer" )
      Coil( #State."Ready For Transfer" )
   END_RUNG
   RUNG wire#w1
      I_Contact( #State."Ready For Transfer Ena" )
      R_Coil( #Cmd."Ready For Transfer" )
   END_RUNG
   // the same network as SCL:
   #State."Ready For Transfer Ena" := #AlwaysON AND NOT #State."Tank LL" AND NOT #State."Dose On Prog" AND NOT #State."CIP Tank" AND NOT #State."CIP Line";
   #State."Ready For Transfer" := #AlwaysON AND #State."Ready For Transfer Ena" AND #Cmd."Ready For Transfer";
   IF #AlwaysON AND NOT #State."Ready For Transfer Ena" THEN #Cmd."Ready For Transfer" := FALSE; END_IF;
END_REGION

REGION Network 9: Buffer Tank Request
   RUNG wire#powerrail
      Contact( #AlwaysON )
      Contact( #State."Ready For Transfer" )
      wire#w1
      Contact( #"BFT-1 Prod Req" )
      wire#w2
      I_Contact( #"Transfer 1 Busy" )
      wire#w3
      I_Contact( #State."BFT-2 EN" )
      I_Contact( #State."BFT-3 EN" )
      Coil( #State."BFT-1 EN" )
   END_RUNG
   RUNG wire#w2
      Contact( #State."BFT-1 EN" )
   END_RUNG wire#w3
   RUNG wire#w1
      Contact( #"BFT-2 Prod Req" )
      wire#w4
      I_Contact( #"Transfer 2 Busy" )
      wire#w5
      I_Contact( #State."BFT-1 EN" )
      I_Contact( #State."BFT-3 EN" )
      Coil( #State."BFT-2 EN" )
   END_RUNG
   RUNG wire#w4
      Contact( #State."BFT-2 EN" )
   END_RUNG wire#w5
   RUNG wire#w1
      Contact( #"BFT-3 Prod Req" )
      wire#w6
      I_Contact( #"Transfer 3 Busy" )
      wire#w7
      I_Contact( #State."BFT-1 EN" )
      I_Contact( #State."BFT-2 EN" )
      Coil( #State."BFT-3 EN" )
   END_RUNG
   RUNG wire#w6
      Contact( #State."BFT-3 EN" )
   END_RUNG wire#w7
   // the same network as SCL:
   #_w1 := #AlwaysON AND #State."Ready For Transfer";
   #State."BFT-1 EN" := #_w1 AND #"BFT-1 Prod Req" AND (NOT #"Transfer 1 Busy" OR #State."BFT-1 EN") AND NOT #State."BFT-2 EN" AND NOT #State."BFT-3 EN";
   #State."BFT-2 EN" := #_w1 AND #"BFT-2 Prod Req" AND (NOT #"Transfer 2 Busy" OR #State."BFT-2 EN") AND NOT #State."BFT-1 EN" AND NOT #State."BFT-3 EN";
   #State."BFT-3 EN" := #_w1 AND #"BFT-3 Prod Req" AND (NOT #"Transfer 3 Busy" OR #State."BFT-3 EN") AND NOT #State."BFT-1 EN" AND NOT #State."BFT-2 EN";
END_REGION

REGION Network 10: Buffer Tank Transfer Progress
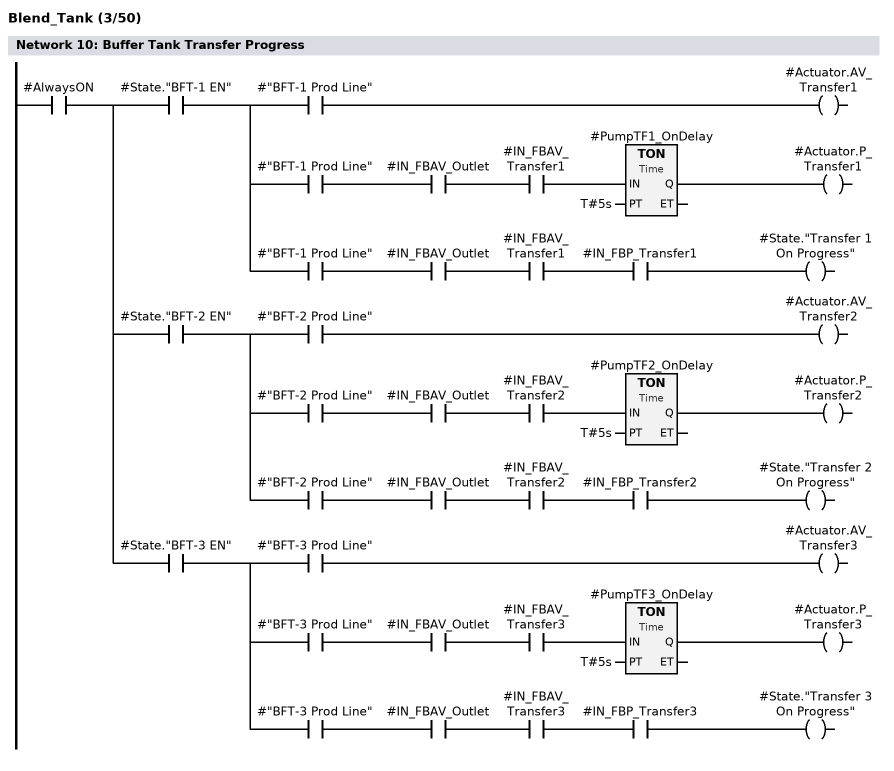
   RUNG wire#powerrail
      Contact( #AlwaysON )
      wire#w1
      Contact( #State."BFT-1 EN" )
      wire#w2
      Contact( #"BFT-1 Prod Line" )
      Coil( #Actuator.AV_Transfer1 )
   END_RUNG
   RUNG wire#w2
      Contact( #"BFT-1 Prod Line" )
      Contact( #IN_FBAV_Outlet )
      Contact( #IN_FBAV_Transfer1 )
      { S7_Templates := "time_type := Time" } #PumpTF1_OnDelay.TON(pt := T#5s, et =>)
      Coil( #Actuator.P_Transfer1 )
   END_RUNG
   RUNG wire#w2
      Contact( #"BFT-1 Prod Line" )
      Contact( #IN_FBAV_Outlet )
      Contact( #IN_FBAV_Transfer1 )
      Contact( #IN_FBP_Transfer1 )
      Coil( #State."Transfer 1 On Progress" )
   END_RUNG
   RUNG wire#w1
      Contact( #State."BFT-2 EN" )
      wire#w3
      Contact( #"BFT-2 Prod Line" )
      Coil( #Actuator.AV_Transfer2 )
   END_RUNG
   RUNG wire#w3
      Contact( #"BFT-2 Prod Line" )
      Contact( #IN_FBAV_Outlet )
      Contact( #IN_FBAV_Transfer2 )
      { S7_Templates := "time_type := Time" } #PumpTF2_OnDelay.TON(pt := T#5s, et =>)
      Coil( #Actuator.P_Transfer2 )
   END_RUNG
   RUNG wire#w3
      Contact( #"BFT-2 Prod Line" )
      Contact( #IN_FBAV_Outlet )
      Contact( #IN_FBAV_Transfer2 )
      Contact( #IN_FBP_Transfer2 )
      Coil( #State."Transfer 2 On Progress" )
   END_RUNG
   RUNG wire#w1
      Contact( #State."BFT-3 EN" )
      wire#w4
      Contact( #"BFT-3 Prod Line" )
      Coil( #Actuator.AV_Transfer3 )
   END_RUNG
   RUNG wire#w4
      Contact( #"BFT-3 Prod Line" )
      Contact( #IN_FBAV_Outlet )
      Contact( #IN_FBAV_Transfer3 )
      { S7_Templates := "time_type := Time" } #PumpTF3_OnDelay.TON(pt := T#5s, et =>)
      Coil( #Actuator.P_Transfer3 )
   END_RUNG
   RUNG wire#w4
      Contact( #"BFT-3 Prod Line" )
      Contact( #IN_FBAV_Outlet )
      Contact( #IN_FBAV_Transfer3 )
      Contact( #IN_FBP_Transfer3 )
      Coil( #State."Transfer 3 On Progress" )
   END_RUNG
   // the same network as SCL:
   #_w1 := #AlwaysON AND #State."BFT-1 EN";
   #Actuator.AV_Transfer1 := #_w1 AND #"BFT-1 Prod Line";
   #PumpTF1_OnDelay(IN := #_w1 AND #"BFT-1 Prod Line" AND #IN_FBAV_Outlet AND #IN_FBAV_Transfer1, PT := T#5s);   // TON
   #Actuator.P_Transfer1 := #PumpTF1_OnDelay.Q;
   #State."Transfer 1 On Progress" := #_w1 AND #"BFT-1 Prod Line" AND #IN_FBAV_Outlet AND #IN_FBAV_Transfer1 AND #IN_FBP_Transfer1;
   #_w2 := #AlwaysON AND #State."BFT-2 EN";
   #Actuator.AV_Transfer2 := #_w2 AND #"BFT-2 Prod Line";
   #PumpTF2_OnDelay(IN := #_w2 AND #"BFT-2 Prod Line" AND #IN_FBAV_Outlet AND #IN_FBAV_Transfer2, PT := T#5s);   // TON
   #Actuator.P_Transfer2 := #PumpTF2_OnDelay.Q;
   #State."Transfer 2 On Progress" := #_w2 AND #"BFT-2 Prod Line" AND #IN_FBAV_Outlet AND #IN_FBAV_Transfer2 AND #IN_FBP_Transfer2;
   #_w3 := #AlwaysON AND #State."BFT-3 EN";
   #Actuator.AV_Transfer3 := #_w3 AND #"BFT-3 Prod Line";
   #PumpTF3_OnDelay(IN := #_w3 AND #"BFT-3 Prod Line" AND #IN_FBAV_Outlet AND #IN_FBAV_Transfer3, PT := T#5s);   // TON
   #Actuator.P_Transfer3 := #PumpTF3_OnDelay.Q;
   #State."Transfer 3 On Progress" := #_w3 AND #"BFT-3 Prod Line" AND #IN_FBAV_Outlet AND #IN_FBAV_Transfer3 AND #IN_FBP_Transfer3;
END_REGION

REGION Network 12: Command CIP
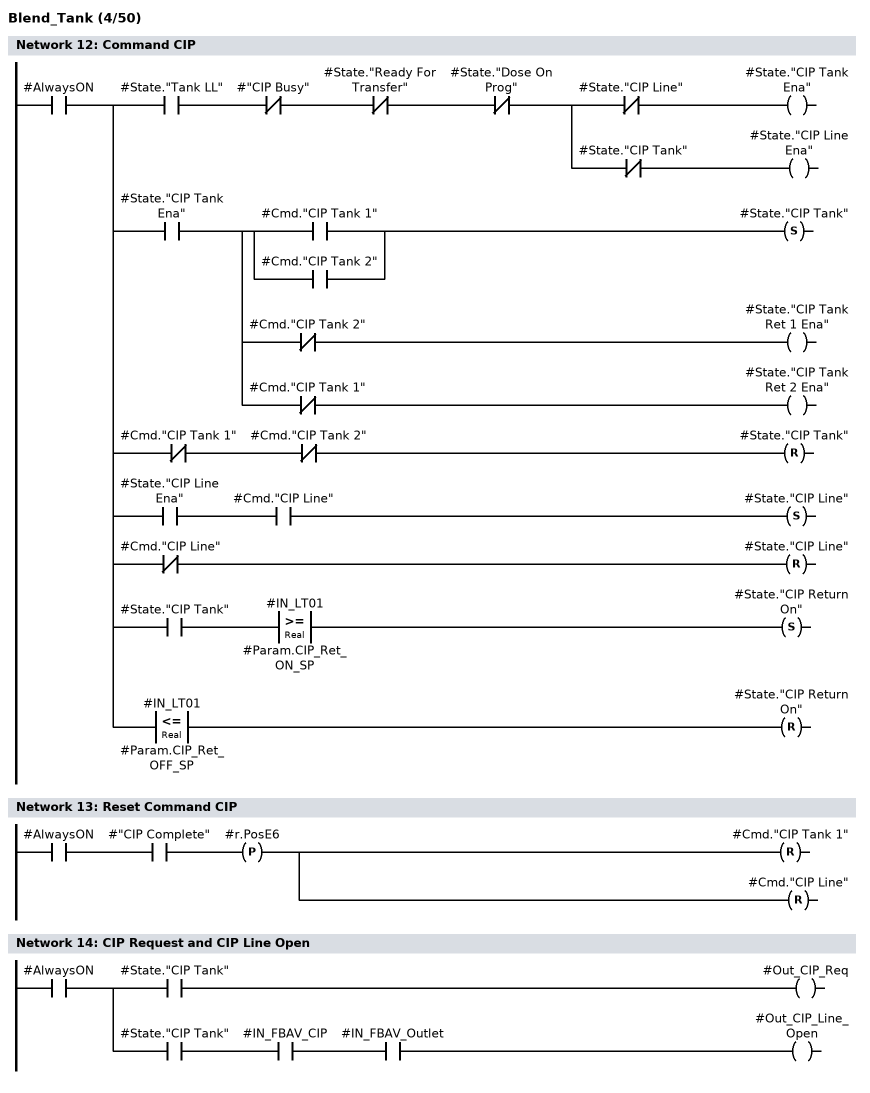
   RUNG wire#powerrail
      Contact( #AlwaysON )
      wire#w1
      Contact( #State."Tank LL" )
      I_Contact( #"CIP Busy" )
      I_Contact( #State."Ready For Transfer" )
      I_Contact( #State."Dose On Prog" )
      wire#w2
      I_Contact( #State."CIP Line" )
      Coil( #State."CIP Tank Ena" )
   END_RUNG
   RUNG wire#w2
      I_Contact( #State."CIP Tank" )
      Coil( #State."CIP Line Ena" )
   END_RUNG
   RUNG wire#w1
      Contact( #State."CIP Tank Ena" )
      wire#w3
      Contact( #Cmd."CIP Tank 1" )
      wire#w4
      S_Coil( #State."CIP Tank" )
   END_RUNG
   RUNG wire#w3
      Contact( #Cmd."CIP Tank 2" )
   END_RUNG wire#w4
   RUNG wire#w3
      I_Contact( #Cmd."CIP Tank 2" )
      Coil( #State."CIP Tank Ret 1 Ena" )
   END_RUNG
   RUNG wire#w3
      I_Contact( #Cmd."CIP Tank 1" )
      Coil( #State."CIP Tank Ret 2 Ena" )
   END_RUNG
   RUNG wire#w1
      I_Contact( #Cmd."CIP Tank 1" )
      I_Contact( #Cmd."CIP Tank 2" )
      R_Coil( #State."CIP Tank" )
   END_RUNG
   RUNG wire#w1
      Contact( #State."CIP Line Ena" )
      Contact( #Cmd."CIP Line" )
      S_Coil( #State."CIP Line" )
   END_RUNG
   RUNG wire#w1
      I_Contact( #Cmd."CIP Line" )
      R_Coil( #State."CIP Line" )
   END_RUNG
   RUNG wire#w1
      Contact( #State."CIP Tank" )
      { S7_Templates := "SrcType := Real" } GE_Contact(in1 := #IN_LT01, in2 := #Param.CIP_Ret_ON_SP)
      S_Coil( #State."CIP Return On" )
   END_RUNG
   RUNG wire#w1
      { S7_Templates := "SrcType := Real" } LE_Contact(in1 := #IN_LT01, in2 := #Param.CIP_Ret_OFF_SP)
      R_Coil( #State."CIP Return On" )
   END_RUNG
   // the same network as SCL:
   #_w1 := #AlwaysON AND #State."Tank LL" AND NOT #"CIP Busy" AND NOT #State."Ready For Transfer" AND NOT #State."Dose On Prog";
   #State."CIP Tank Ena" := #_w1 AND NOT #State."CIP Line";
   #State."CIP Line Ena" := #_w1 AND NOT #State."CIP Tank";
   #_w2 := #AlwaysON AND #State."CIP Tank Ena";
   IF #_w2 AND (#Cmd."CIP Tank 1" OR #Cmd."CIP Tank 2") THEN #State."CIP Tank" := TRUE; END_IF;
   #State."CIP Tank Ret 1 Ena" := #_w2 AND NOT #Cmd."CIP Tank 2";
   #State."CIP Tank Ret 2 Ena" := #_w2 AND NOT #Cmd."CIP Tank 1";
   IF #AlwaysON AND NOT #Cmd."CIP Tank 1" AND NOT #Cmd."CIP Tank 2" THEN #State."CIP Tank" := FALSE; END_IF;
   IF #AlwaysON AND #State."CIP Line Ena" AND #Cmd."CIP Line" THEN #State."CIP Line" := TRUE; END_IF;
   IF #AlwaysON AND NOT #Cmd."CIP Line" THEN #State."CIP Line" := FALSE; END_IF;
   IF #AlwaysON AND #State."CIP Tank" AND (#IN_LT01 >= #Param.CIP_Ret_ON_SP) THEN
       #State."CIP Return On" := TRUE;
   END_IF;
   IF #AlwaysON AND (#IN_LT01 <= #Param.CIP_Ret_OFF_SP) THEN #State."CIP Return On" := FALSE; END_IF;
END_REGION

REGION Network 13: Reset Command CIP
   RUNG wire#powerrail
      Contact( #AlwaysON )
      Contact( #"CIP Complete" )
      P_Trig( #r.PosE6 )
      wire#w1
      R_Coil( #Cmd."CIP Tank 1" )
   END_RUNG
   RUNG wire#w1
      R_Coil( #Cmd."CIP Line" )
   END_RUNG
   // the same network as SCL:
   #_w1 := #AlwaysON AND #"CIP Complete";
   #_w2 := #_w1 AND NOT #r.PosE6;   // rising edge
   #r.PosE6 := #_w1;
   IF #_w2 THEN
       #Cmd."CIP Tank 1" := FALSE;
       #Cmd."CIP Line" := FALSE;
   END_IF;
END_REGION

REGION Network 14: CIP Request and CIP Line Open
   RUNG wire#powerrail
      Contact( #AlwaysON )
      wire#w1
      Contact( #State."CIP Tank" )
      Coil( #Out_CIP_Req )
   END_RUNG
   RUNG wire#w1
      Contact( #State."CIP Tank" )
      Contact( #IN_FBAV_CIP )
      Contact( #IN_FBAV_Outlet )
      Coil( #Out_CIP_Line_Open )
   END_RUNG
   // the same network as SCL:
   #Out_CIP_Req := #AlwaysON AND #State."CIP Tank";
   #Out_CIP_Line_Open := #AlwaysON AND #State."CIP Tank" AND #IN_FBAV_CIP AND #IN_FBAV_Outlet;
END_REGION

